ABB RAPID module: hersheyCursiveModule.mod

MODULE hersheyCursiveModule
  ! Character: a
  PROC char_a()
    VAR robtarget pTarget;
    pTarget := refTarget;
    pTarget.trans := [9,17.0,0];
    MoveL pTarget,vSpeed,fine,tTool\WObj:=wWobj;
    Set do_pen;
    pTarget.trans := [8,19.0,0];
    MoveL pTarget,vSpeed,z0,tTool\WObj:=wWobj;
    pTarget.trans := [6,20.0,0];
    MoveL pTarget,vSpeed,z0,tTool\WObj:=wWobj;
    pTarget.trans := [4,20.0,0];
    MoveL pTarget,vSpeed,z0,tTool\WObj:=wWobj;
    pTarget.trans := [2,19.0,0];
    MoveL pTarget,vSpeed,z0,tTool\WObj:=wWobj;
    pTarget.trans := [1,18.0,0];
    MoveL pTarget,vSpeed,z0,tTool\WObj:=wWobj;
    pTarget.trans := [0,16.0,0];
    MoveL pTarget,vSpeed,z0,tTool\WObj:=wWobj;
    pTarget.trans := [0,14.0,0];
    MoveL pTarget,vSpeed,z0,tTool\WObj:=wWobj;
    pTarget.trans := [1,12.0,0];
    MoveL pTarget,vSpeed,z0,tTool\WObj:=wWobj;
    pTarget.trans := [3,11.0,0];
    MoveL pTarget,vSpeed,z0,tTool\WObj:=wWobj;
    pTarget.trans := [5,11.0,0];
    MoveL pTarget,vSpeed,z0,tTool\WObj:=wWobj;
    pTarget.trans := [7,12.0,0];
    MoveL pTarget,vSpeed,z0,tTool\WObj:=wWobj;
    pTarget.trans := [8,14.0,0];
    MoveL pTarget,vSpeed,z0,tTool\WObj:=wWobj;
    pTarget.trans := [10,20.0,0];
    MoveL pTarget,vSpeed,z0,tTool\WObj:=wWobj;
    pTarget.trans := [9,15.0,0];
    MoveL pTarget,vSpeed,z0,tTool\WObj:=wWobj;
    pTarget.trans := [9,12.0,0];
    MoveL pTarget,vSpeed,z0,tTool\WObj:=wWobj;
    pTarget.trans := [10,11.0,0];
    MoveL pTarget,vSpeed,z0,tTool\WObj:=wWobj;
    pTarget.trans := [11,11.0,0];
    MoveL pTarget,vSpeed,z0,tTool\WObj:=wWobj;
    pTarget.trans := [13,12.0,0];
    MoveL pTarget,vSpeed,z0,tTool\WObj:=wWobj;
    pTarget.trans := [14,13.0,0];
    MoveL pTarget,vSpeed,z0,tTool\WObj:=wWobj;
    pTarget.trans := [16,16.0,0];
    MoveL pTarget,vSpeed,fine,tTool\WObj:=wWobj;
    Reset do_pen;
    MoveL RelTool(pTarget,0,0,-2),vSpeed,z0,tTool\WObj:=wWobj;
    wWobj.oframe.trans.x := wWobj.oframe.trans.x + 16;
ENDPROC
  ! Character: b
  PROC char_b()
    VAR robtarget pTarget;
    pTarget := refTarget;
    pTarget.trans := [0,16.0,0];
    MoveL pTarget,vSpeed,fine,tTool\WObj:=wWobj;
    Set do_pen;
    pTarget.trans := [2,19.0,0];
    MoveL pTarget,vSpeed,z0,tTool\WObj:=wWobj;
    pTarget.trans := [5,24.0,0];
    MoveL pTarget,vSpeed,z0,tTool\WObj:=wWobj;
    pTarget.trans := [6,26.0,0];
    MoveL pTarget,vSpeed,z0,tTool\WObj:=wWobj;
    pTarget.trans := [7,29.0,0];
    MoveL pTarget,vSpeed,z0,tTool\WObj:=wWobj;
    pTarget.trans := [7,31.0,0];
    MoveL pTarget,vSpeed,z0,tTool\WObj:=wWobj;
    pTarget.trans := [6,32.0,0];
    MoveL pTarget,vSpeed,z0,tTool\WObj:=wWobj;
    pTarget.trans := [4,31.0,0];
    MoveL pTarget,vSpeed,z0,tTool\WObj:=wWobj;
    pTarget.trans := [3,29.0,0];
    MoveL pTarget,vSpeed,z0,tTool\WObj:=wWobj;
    pTarget.trans := [2,25.0,0];
    MoveL pTarget,vSpeed,z0,tTool\WObj:=wWobj;
    pTarget.trans := [1,18.0,0];
    MoveL pTarget,vSpeed,z0,tTool\WObj:=wWobj;
    pTarget.trans := [1,12.0,0];
    MoveL pTarget,vSpeed,z0,tTool\WObj:=wWobj;
    pTarget.trans := [2,11.0,0];
    MoveL pTarget,vSpeed,z0,tTool\WObj:=wWobj;
    pTarget.trans := [3,11.0,0];
    MoveL pTarget,vSpeed,z0,tTool\WObj:=wWobj;
    pTarget.trans := [5,12.0,0];
    MoveL pTarget,vSpeed,z0,tTool\WObj:=wWobj;
    pTarget.trans := [7,14.0,0];
    MoveL pTarget,vSpeed,z0,tTool\WObj:=wWobj;
    pTarget.trans := [8,17.0,0];
    MoveL pTarget,vSpeed,z0,tTool\WObj:=wWobj;
    pTarget.trans := [8,20.0,0];
    MoveL pTarget,vSpeed,z0,tTool\WObj:=wWobj;
    pTarget.trans := [9,16.0,0];
    MoveL pTarget,vSpeed,z0,tTool\WObj:=wWobj;
    pTarget.trans := [10,15.0,0];
    MoveL pTarget,vSpeed,z0,tTool\WObj:=wWobj;
    pTarget.trans := [12,15.0,0];
    MoveL pTarget,vSpeed,z0,tTool\WObj:=wWobj;
    pTarget.trans := [14,16.0,0];
    MoveL pTarget,vSpeed,fine,tTool\WObj:=wWobj;
    Reset do_pen;
    MoveL RelTool(pTarget,0,0,-2),vSpeed,z0,tTool\WObj:=wWobj;
    wWobj.oframe.trans.x := wWobj.oframe.trans.x + 14;
ENDPROC
  ! Character: c
  PROC char_c()
    VAR robtarget pTarget;
    pTarget := refTarget;
    pTarget.trans := [7,18.0,0];
    MoveL pTarget,vSpeed,fine,tTool\WObj:=wWobj;
    Set do_pen;
    pTarget.trans := [7,19.0,0];
    MoveL pTarget,vSpeed,z0,tTool\WObj:=wWobj;
    pTarget.trans := [6,20.0,0];
    MoveL pTarget,vSpeed,z0,tTool\WObj:=wWobj;
    pTarget.trans := [4,20.0,0];
    MoveL pTarget,vSpeed,z0,tTool\WObj:=wWobj;
    pTarget.trans := [2,19.0,0];
    MoveL pTarget,vSpeed,z0,tTool\WObj:=wWobj;
    pTarget.trans := [1,18.0,0];
    MoveL pTarget,vSpeed,z0,tTool\WObj:=wWobj;
    pTarget.trans := [0,16.0,0];
    MoveL pTarget,vSpeed,z0,tTool\WObj:=wWobj;
    pTarget.trans := [0,14.0,0];
    MoveL pTarget,vSpeed,z0,tTool\WObj:=wWobj;
    pTarget.trans := [1,12.0,0];
    MoveL pTarget,vSpeed,z0,tTool\WObj:=wWobj;
    pTarget.trans := [3,11.0,0];
    MoveL pTarget,vSpeed,z0,tTool\WObj:=wWobj;
    pTarget.trans := [6,11.0,0];
    MoveL pTarget,vSpeed,z0,tTool\WObj:=wWobj;
    pTarget.trans := [9,13.0,0];
    MoveL pTarget,vSpeed,z0,tTool\WObj:=wWobj;
    pTarget.trans := [11,16.0,0];
    MoveL pTarget,vSpeed,fine,tTool\WObj:=wWobj;
    Reset do_pen;
    MoveL RelTool(pTarget,0,0,-2),vSpeed,z0,tTool\WObj:=wWobj;
    wWobj.oframe.trans.x := wWobj.oframe.trans.x + 11;
ENDPROC
  ! Character: d
  PROC char_d()
    VAR robtarget pTarget;
    pTarget := refTarget;
    pTarget.trans := [9,17.0,0];
    MoveL pTarget,vSpeed,fine,tTool\WObj:=wWobj;
    Set do_pen;
    pTarget.trans := [8,19.0,0];
    MoveL pTarget,vSpeed,z0,tTool\WObj:=wWobj;
    pTarget.trans := [6,20.0,0];
    MoveL pTarget,vSpeed,z0,tTool\WObj:=wWobj;
    pTarget.trans := [4,20.0,0];
    MoveL pTarget,vSpeed,z0,tTool\WObj:=wWobj;
    pTarget.trans := [2,19.0,0];
    MoveL pTarget,vSpeed,z0,tTool\WObj:=wWobj;
    pTarget.trans := [1,18.0,0];
    MoveL pTarget,vSpeed,z0,tTool\WObj:=wWobj;
    pTarget.trans := [0,16.0,0];
    MoveL pTarget,vSpeed,z0,tTool\WObj:=wWobj;
    pTarget.trans := [0,14.0,0];
    MoveL pTarget,vSpeed,z0,tTool\WObj:=wWobj;
    pTarget.trans := [1,12.0,0];
    MoveL pTarget,vSpeed,z0,tTool\WObj:=wWobj;
    pTarget.trans := [3,11.0,0];
    MoveL pTarget,vSpeed,z0,tTool\WObj:=wWobj;
    pTarget.trans := [5,11.0,0];
    MoveL pTarget,vSpeed,z0,tTool\WObj:=wWobj;
    pTarget.trans := [7,12.0,0];
    MoveL pTarget,vSpeed,z0,tTool\WObj:=wWobj;
    pTarget.trans := [8,14.0,0];
    MoveL pTarget,vSpeed,z0,tTool\WObj:=wWobj;
    pTarget.trans := [14,32.0,0];
    MoveL pTarget,vSpeed,fine,tTool\WObj:=wWobj;
    Reset do_pen;
    MoveL RelTool(pTarget,0,0,-2),vSpeed,z0,tTool\WObj:=wWobj;
    pTarget.trans := [10,20.0,0];
    MoveL pTarget,vSpeed,fine,tTool\WObj:=wWobj;
    Set do_pen;
    pTarget.trans := [9,15.0,0];
    MoveL pTarget,vSpeed,z0,tTool\WObj:=wWobj;
    pTarget.trans := [9,12.0,0];
    MoveL pTarget,vSpeed,z0,tTool\WObj:=wWobj;
    pTarget.trans := [10,11.0,0];
    MoveL pTarget,vSpeed,z0,tTool\WObj:=wWobj;
    pTarget.trans := [11,11.0,0];
    MoveL pTarget,vSpeed,z0,tTool\WObj:=wWobj;
    pTarget.trans := [13,12.0,0];
    MoveL pTarget,vSpeed,z0,tTool\WObj:=wWobj;
    pTarget.trans := [14,13.0,0];
    MoveL pTarget,vSpeed,z0,tTool\WObj:=wWobj;
    pTarget.trans := [16,16.0,0];
    MoveL pTarget,vSpeed,fine,tTool\WObj:=wWobj;
    Reset do_pen;
    MoveL RelTool(pTarget,0,0,-2),vSpeed,z0,tTool\WObj:=wWobj;
    wWobj.oframe.trans.x := wWobj.oframe.trans.x + 16;
ENDPROC
  ! Character: e
  PROC char_e()
    VAR robtarget pTarget;
    pTarget := refTarget;
    pTarget.trans := [1,13.0,0];
    MoveL pTarget,vSpeed,fine,tTool\WObj:=wWobj;
    Set do_pen;
    pTarget.trans := [3,14.0,0];
    MoveL pTarget,vSpeed,z0,tTool\WObj:=wWobj;
    pTarget.trans := [4,15.0,0];
    MoveL pTarget,vSpeed,z0,tTool\WObj:=wWobj;
    pTarget.trans := [5,17.0,0];
    MoveL pTarget,vSpeed,z0,tTool\WObj:=wWobj;
    pTarget.trans := [5,19.0,0];
    MoveL pTarget,vSpeed,z0,tTool\WObj:=wWobj;
    pTarget.trans := [4,20.0,0];
    MoveL pTarget,vSpeed,z0,tTool\WObj:=wWobj;
    pTarget.trans := [3,20.0,0];
    MoveL pTarget,vSpeed,z0,tTool\WObj:=wWobj;
    pTarget.trans := [1,19.0,0];
    MoveL pTarget,vSpeed,z0,tTool\WObj:=wWobj;
    pTarget.trans := [0,17.0,0];
    MoveL pTarget,vSpeed,z0,tTool\WObj:=wWobj;
    pTarget.trans := [0,14.0,0];
    MoveL pTarget,vSpeed,z0,tTool\WObj:=wWobj;
    pTarget.trans := [1,12.0,0];
    MoveL pTarget,vSpeed,z0,tTool\WObj:=wWobj;
    pTarget.trans := [3,11.0,0];
    MoveL pTarget,vSpeed,z0,tTool\WObj:=wWobj;
    pTarget.trans := [5,11.0,0];
    MoveL pTarget,vSpeed,z0,tTool\WObj:=wWobj;
    pTarget.trans := [7,12.0,0];
    MoveL pTarget,vSpeed,z0,tTool\WObj:=wWobj;
    pTarget.trans := [8,13.0,0];
    MoveL pTarget,vSpeed,z0,tTool\WObj:=wWobj;
    pTarget.trans := [10,16.0,0];
    MoveL pTarget,vSpeed,fine,tTool\WObj:=wWobj;
    Reset do_pen;
    MoveL RelTool(pTarget,0,0,-2),vSpeed,z0,tTool\WObj:=wWobj;
    wWobj.oframe.trans.x := wWobj.oframe.trans.x + 10;
ENDPROC
  ! Character: f
  PROC char_f()
    VAR robtarget pTarget;
    pTarget := refTarget;
    pTarget.trans := [0,16.0,0];
    MoveL pTarget,vSpeed,fine,tTool\WObj:=wWobj;
    Set do_pen;
    pTarget.trans := [4,21.0,0];
    MoveL pTarget,vSpeed,z0,tTool\WObj:=wWobj;
    pTarget.trans := [6,24.0,0];
    MoveL pTarget,vSpeed,z0,tTool\WObj:=wWobj;
    pTarget.trans := [7,26.0,0];
    MoveL pTarget,vSpeed,z0,tTool\WObj:=wWobj;
    pTarget.trans := [8,29.0,0];
    MoveL pTarget,vSpeed,z0,tTool\WObj:=wWobj;
    pTarget.trans := [8,31.0,0];
    MoveL pTarget,vSpeed,z0,tTool\WObj:=wWobj;
    pTarget.trans := [7,32.0,0];
    MoveL pTarget,vSpeed,z0,tTool\WObj:=wWobj;
    pTarget.trans := [5,31.0,0];
    MoveL pTarget,vSpeed,z0,tTool\WObj:=wWobj;
    pTarget.trans := [4,29.0,0];
    MoveL pTarget,vSpeed,z0,tTool\WObj:=wWobj;
    pTarget.trans := [2,21.0,0];
    MoveL pTarget,vSpeed,z0,tTool\WObj:=wWobj;
    pTarget.trans := [-1,12.0,0];
    MoveL pTarget,vSpeed,z0,tTool\WObj:=wWobj;
    pTarget.trans := [-4,5.0,0];
    MoveL pTarget,vSpeed,z0,tTool\WObj:=wWobj;
    pTarget.trans := [-5,2.0,0];
    MoveL pTarget,vSpeed,z0,tTool\WObj:=wWobj;
    pTarget.trans := [-5,0.0,0];
    MoveL pTarget,vSpeed,z0,tTool\WObj:=wWobj;
    pTarget.trans := [-4,-1.0,0];
    MoveL pTarget,vSpeed,z0,tTool\WObj:=wWobj;
    pTarget.trans := [-2,0.0,0];
    MoveL pTarget,vSpeed,z0,tTool\WObj:=wWobj;
    pTarget.trans := [-1,3.0,0];
    MoveL pTarget,vSpeed,z0,tTool\WObj:=wWobj;
    pTarget.trans := [0,12.0,0];
    MoveL pTarget,vSpeed,z0,tTool\WObj:=wWobj;
    pTarget.trans := [1,11.0,0];
    MoveL pTarget,vSpeed,z0,tTool\WObj:=wWobj;
    pTarget.trans := [3,11.0,0];
    MoveL pTarget,vSpeed,z0,tTool\WObj:=wWobj;
    pTarget.trans := [5,12.0,0];
    MoveL pTarget,vSpeed,z0,tTool\WObj:=wWobj;
    pTarget.trans := [6,13.0,0];
    MoveL pTarget,vSpeed,z0,tTool\WObj:=wWobj;
    pTarget.trans := [8,16.0,0];
    MoveL pTarget,vSpeed,fine,tTool\WObj:=wWobj;
    Reset do_pen;
    MoveL RelTool(pTarget,0,0,-2),vSpeed,z0,tTool\WObj:=wWobj;
    wWobj.oframe.trans.x := wWobj.oframe.trans.x + 13;
ENDPROC
  ! Character: g
  PROC char_g()
    VAR robtarget pTarget;
    pTarget := refTarget;
    pTarget.trans := [9,17.0,0];
    MoveL pTarget,vSpeed,fine,tTool\WObj:=wWobj;
    Set do_pen;
    pTarget.trans := [8,19.0,0];
    MoveL pTarget,vSpeed,z0,tTool\WObj:=wWobj;
    pTarget.trans := [6,20.0,0];
    MoveL pTarget,vSpeed,z0,tTool\WObj:=wWobj;
    pTarget.trans := [4,20.0,0];
    MoveL pTarget,vSpeed,z0,tTool\WObj:=wWobj;
    pTarget.trans := [2,19.0,0];
    MoveL pTarget,vSpeed,z0,tTool\WObj:=wWobj;
    pTarget.trans := [1,18.0,0];
    MoveL pTarget,vSpeed,z0,tTool\WObj:=wWobj;
    pTarget.trans := [0,16.0,0];
    MoveL pTarget,vSpeed,z0,tTool\WObj:=wWobj;
    pTarget.trans := [0,14.0,0];
    MoveL pTarget,vSpeed,z0,tTool\WObj:=wWobj;
    pTarget.trans := [1,12.0,0];
    MoveL pTarget,vSpeed,z0,tTool\WObj:=wWobj;
    pTarget.trans := [3,11.0,0];
    MoveL pTarget,vSpeed,z0,tTool\WObj:=wWobj;
    pTarget.trans := [5,11.0,0];
    MoveL pTarget,vSpeed,z0,tTool\WObj:=wWobj;
    pTarget.trans := [7,12.0,0];
    MoveL pTarget,vSpeed,z0,tTool\WObj:=wWobj;
    pTarget.trans := [8,13.0,0];
    MoveL pTarget,vSpeed,fine,tTool\WObj:=wWobj;
    Reset do_pen;
    MoveL RelTool(pTarget,0,0,-2),vSpeed,z0,tTool\WObj:=wWobj;
    pTarget.trans := [10,20.0,0];
    MoveL pTarget,vSpeed,fine,tTool\WObj:=wWobj;
    Set do_pen;
    pTarget.trans := [8,13.0,0];
    MoveL pTarget,vSpeed,z0,tTool\WObj:=wWobj;
    pTarget.trans := [4,2.0,0];
    MoveL pTarget,vSpeed,z0,tTool\WObj:=wWobj;
    pTarget.trans := [3,0.0,0];
    MoveL pTarget,vSpeed,z0,tTool\WObj:=wWobj;
    pTarget.trans := [1,-1.0,0];
    MoveL pTarget,vSpeed,z0,tTool\WObj:=wWobj;
    pTarget.trans := [0,0.0,0];
    MoveL pTarget,vSpeed,z0,tTool\WObj:=wWobj;
    pTarget.trans := [0,2.0,0];
    MoveL pTarget,vSpeed,z0,tTool\WObj:=wWobj;
    pTarget.trans := [1,5.0,0];
    MoveL pTarget,vSpeed,z0,tTool\WObj:=wWobj;
    pTarget.trans := [4,8.0,0];
    MoveL pTarget,vSpeed,z0,tTool\WObj:=wWobj;
    pTarget.trans := [7,10.0,0];
    MoveL pTarget,vSpeed,z0,tTool\WObj:=wWobj;
    pTarget.trans := [9,11.0,0];
    MoveL pTarget,vSpeed,z0,tTool\WObj:=wWobj;
    pTarget.trans := [12,13.0,0];
    MoveL pTarget,vSpeed,z0,tTool\WObj:=wWobj;
    pTarget.trans := [15,16.0,0];
    MoveL pTarget,vSpeed,fine,tTool\WObj:=wWobj;
    Reset do_pen;
    MoveL RelTool(pTarget,0,0,-2),vSpeed,z0,tTool\WObj:=wWobj;
    wWobj.oframe.trans.x := wWobj.oframe.trans.x + 15;
ENDPROC
  ! Character: h
  PROC char_h()
    VAR robtarget pTarget;
    pTarget := refTarget;
    pTarget.trans := [0,16.0,0];
    MoveL pTarget,vSpeed,fine,tTool\WObj:=wWobj;
    Set do_pen;
    pTarget.trans := [2,19.0,0];
    MoveL pTarget,vSpeed,z0,tTool\WObj:=wWobj;
    pTarget.trans := [5,24.0,0];
    MoveL pTarget,vSpeed,z0,tTool\WObj:=wWobj;
    pTarget.trans := [6,26.0,0];
    MoveL pTarget,vSpeed,z0,tTool\WObj:=wWobj;
    pTarget.trans := [7,29.0,0];
    MoveL pTarget,vSpeed,z0,tTool\WObj:=wWobj;
    pTarget.trans := [7,31.0,0];
    MoveL pTarget,vSpeed,z0,tTool\WObj:=wWobj;
    pTarget.trans := [6,32.0,0];
    MoveL pTarget,vSpeed,z0,tTool\WObj:=wWobj;
    pTarget.trans := [4,31.0,0];
    MoveL pTarget,vSpeed,z0,tTool\WObj:=wWobj;
    pTarget.trans := [3,29.0,0];
    MoveL pTarget,vSpeed,z0,tTool\WObj:=wWobj;
    pTarget.trans := [2,25.0,0];
    MoveL pTarget,vSpeed,z0,tTool\WObj:=wWobj;
    pTarget.trans := [1,19.0,0];
    MoveL pTarget,vSpeed,z0,tTool\WObj:=wWobj;
    pTarget.trans := [0,11.0,0];
    MoveL pTarget,vSpeed,fine,tTool\WObj:=wWobj;
    Reset do_pen;
    MoveL RelTool(pTarget,0,0,-2),vSpeed,z0,tTool\WObj:=wWobj;
    pTarget.trans := [0,11.0,0];
    MoveL pTarget,vSpeed,fine,tTool\WObj:=wWobj;
    Set do_pen;
    pTarget.trans := [1,14.0,0];
    MoveL pTarget,vSpeed,z0,tTool\WObj:=wWobj;
    pTarget.trans := [2,16.0,0];
    MoveL pTarget,vSpeed,z0,tTool\WObj:=wWobj;
    pTarget.trans := [4,19.0,0];
    MoveL pTarget,vSpeed,z0,tTool\WObj:=wWobj;
    pTarget.trans := [6,20.0,0];
    MoveL pTarget,vSpeed,z0,tTool\WObj:=wWobj;
    pTarget.trans := [8,20.0,0];
    MoveL pTarget,vSpeed,z0,tTool\WObj:=wWobj;
    pTarget.trans := [9,19.0,0];
    MoveL pTarget,vSpeed,z0,tTool\WObj:=wWobj;
    pTarget.trans := [9,17.0,0];
    MoveL pTarget,vSpeed,z0,tTool\WObj:=wWobj;
    pTarget.trans := [8,14.0,0];
    MoveL pTarget,vSpeed,z0,tTool\WObj:=wWobj;
    pTarget.trans := [8,12.0,0];
    MoveL pTarget,vSpeed,z0,tTool\WObj:=wWobj;
    pTarget.trans := [9,11.0,0];
    MoveL pTarget,vSpeed,z0,tTool\WObj:=wWobj;
    pTarget.trans := [10,11.0,0];
    MoveL pTarget,vSpeed,z0,tTool\WObj:=wWobj;
    pTarget.trans := [12,12.0,0];
    MoveL pTarget,vSpeed,z0,tTool\WObj:=wWobj;
    pTarget.trans := [13,13.0,0];
    MoveL pTarget,vSpeed,z0,tTool\WObj:=wWobj;
    pTarget.trans := [15,16.0,0];
    MoveL pTarget,vSpeed,fine,tTool\WObj:=wWobj;
    Reset do_pen;
    MoveL RelTool(pTarget,0,0,-2),vSpeed,z0,tTool\WObj:=wWobj;
    wWobj.oframe.trans.x := wWobj.oframe.trans.x + 15;
ENDPROC
  ! Character: i
  PROC char_i()
    VAR robtarget pTarget;
    pTarget := refTarget;
    pTarget.trans := [3,25.0,0];
    MoveL pTarget,vSpeed,fine,tTool\WObj:=wWobj;
    Set do_pen;
    pTarget.trans := [3,24.0,0];
    MoveL pTarget,vSpeed,z0,tTool\WObj:=wWobj;
    pTarget.trans := [4,24.0,0];
    MoveL pTarget,vSpeed,z0,tTool\WObj:=wWobj;
    pTarget.trans := [4,25.0,0];
    MoveL pTarget,vSpeed,z0,tTool\WObj:=wWobj;
    pTarget.trans := [3,25.0,0];
    MoveL pTarget,vSpeed,fine,tTool\WObj:=wWobj;
    Reset do_pen;
    MoveL RelTool(pTarget,0,0,-2),vSpeed,z0,tTool\WObj:=wWobj;
    pTarget.trans := [0,16.0,0];
    MoveL pTarget,vSpeed,fine,tTool\WObj:=wWobj;
    Set do_pen;
    pTarget.trans := [2,20.0,0];
    MoveL pTarget,vSpeed,z0,tTool\WObj:=wWobj;
    pTarget.trans := [0,14.0,0];
    MoveL pTarget,vSpeed,z0,tTool\WObj:=wWobj;
    pTarget.trans := [0,12.0,0];
    MoveL pTarget,vSpeed,z0,tTool\WObj:=wWobj;
    pTarget.trans := [1,11.0,0];
    MoveL pTarget,vSpeed,z0,tTool\WObj:=wWobj;
    pTarget.trans := [2,11.0,0];
    MoveL pTarget,vSpeed,z0,tTool\WObj:=wWobj;
    pTarget.trans := [4,12.0,0];
    MoveL pTarget,vSpeed,z0,tTool\WObj:=wWobj;
    pTarget.trans := [5,13.0,0];
    MoveL pTarget,vSpeed,z0,tTool\WObj:=wWobj;
    pTarget.trans := [7,16.0,0];
    MoveL pTarget,vSpeed,fine,tTool\WObj:=wWobj;
    Reset do_pen;
    MoveL RelTool(pTarget,0,0,-2),vSpeed,z0,tTool\WObj:=wWobj;
    wWobj.oframe.trans.x := wWobj.oframe.trans.x + 7;
ENDPROC
  ! Character: j
  PROC char_j()
    VAR robtarget pTarget;
    pTarget := refTarget;
    pTarget.trans := [3,25.0,0];
    MoveL pTarget,vSpeed,fine,tTool\WObj:=wWobj;
    Set do_pen;
    pTarget.trans := [3,24.0,0];
    MoveL pTarget,vSpeed,z0,tTool\WObj:=wWobj;
    pTarget.trans := [4,24.0,0];
    MoveL pTarget,vSpeed,z0,tTool\WObj:=wWobj;
    pTarget.trans := [4,25.0,0];
    MoveL pTarget,vSpeed,z0,tTool\WObj:=wWobj;
    pTarget.trans := [3,25.0,0];
    MoveL pTarget,vSpeed,fine,tTool\WObj:=wWobj;
    Reset do_pen;
    MoveL RelTool(pTarget,0,0,-2),vSpeed,z0,tTool\WObj:=wWobj;
    pTarget.trans := [0,16.0,0];
    MoveL pTarget,vSpeed,fine,tTool\WObj:=wWobj;
    Set do_pen;
    pTarget.trans := [2,20.0,0];
    MoveL pTarget,vSpeed,z0,tTool\WObj:=wWobj;
    pTarget.trans := [-4,2.0,0];
    MoveL pTarget,vSpeed,z0,tTool\WObj:=wWobj;
    pTarget.trans := [-5,0.0,0];
    MoveL pTarget,vSpeed,z0,tTool\WObj:=wWobj;
    pTarget.trans := [-7,-1.0,0];
    MoveL pTarget,vSpeed,z0,tTool\WObj:=wWobj;
    pTarget.trans := [-8,0.0,0];
    MoveL pTarget,vSpeed,z0,tTool\WObj:=wWobj;
    pTarget.trans := [-8,2.0,0];
    MoveL pTarget,vSpeed,z0,tTool\WObj:=wWobj;
    pTarget.trans := [-7,5.0,0];
    MoveL pTarget,vSpeed,z0,tTool\WObj:=wWobj;
    pTarget.trans := [-4,8.0,0];
    MoveL pTarget,vSpeed,z0,tTool\WObj:=wWobj;
    pTarget.trans := [-1,10.0,0];
    MoveL pTarget,vSpeed,z0,tTool\WObj:=wWobj;
    pTarget.trans := [1,11.0,0];
    MoveL pTarget,vSpeed,z0,tTool\WObj:=wWobj;
    pTarget.trans := [4,13.0,0];
    MoveL pTarget,vSpeed,z0,tTool\WObj:=wWobj;
    pTarget.trans := [7,16.0,0];
    MoveL pTarget,vSpeed,fine,tTool\WObj:=wWobj;
    Reset do_pen;
    MoveL RelTool(pTarget,0,0,-2),vSpeed,z0,tTool\WObj:=wWobj;
    wWobj.oframe.trans.x := wWobj.oframe.trans.x + 15;
ENDPROC
  ! Character: k
  PROC char_k()
    VAR robtarget pTarget;
    pTarget := refTarget;
    pTarget.trans := [0,16.0,0];
    MoveL pTarget,vSpeed,fine,tTool\WObj:=wWobj;
    Set do_pen;
    pTarget.trans := [2,19.0,0];
    MoveL pTarget,vSpeed,z0,tTool\WObj:=wWobj;
    pTarget.trans := [5,24.0,0];
    MoveL pTarget,vSpeed,z0,tTool\WObj:=wWobj;
    pTarget.trans := [6,26.0,0];
    MoveL pTarget,vSpeed,z0,tTool\WObj:=wWobj;
    pTarget.trans := [7,29.0,0];
    MoveL pTarget,vSpeed,z0,tTool\WObj:=wWobj;
    pTarget.trans := [7,31.0,0];
    MoveL pTarget,vSpeed,z0,tTool\WObj:=wWobj;
    pTarget.trans := [6,32.0,0];
    MoveL pTarget,vSpeed,z0,tTool\WObj:=wWobj;
    pTarget.trans := [4,31.0,0];
    MoveL pTarget,vSpeed,z0,tTool\WObj:=wWobj;
    pTarget.trans := [3,29.0,0];
    MoveL pTarget,vSpeed,z0,tTool\WObj:=wWobj;
    pTarget.trans := [2,25.0,0];
    MoveL pTarget,vSpeed,z0,tTool\WObj:=wWobj;
    pTarget.trans := [1,19.0,0];
    MoveL pTarget,vSpeed,z0,tTool\WObj:=wWobj;
    pTarget.trans := [0,11.0,0];
    MoveL pTarget,vSpeed,fine,tTool\WObj:=wWobj;
    Reset do_pen;
    MoveL RelTool(pTarget,0,0,-2),vSpeed,z0,tTool\WObj:=wWobj;
    pTarget.trans := [0,11.0,0];
    MoveL pTarget,vSpeed,fine,tTool\WObj:=wWobj;
    Set do_pen;
    pTarget.trans := [1,14.0,0];
    MoveL pTarget,vSpeed,z0,tTool\WObj:=wWobj;
    pTarget.trans := [2,16.0,0];
    MoveL pTarget,vSpeed,z0,tTool\WObj:=wWobj;
    pTarget.trans := [4,19.0,0];
    MoveL pTarget,vSpeed,z0,tTool\WObj:=wWobj;
    pTarget.trans := [6,20.0,0];
    MoveL pTarget,vSpeed,z0,tTool\WObj:=wWobj;
    pTarget.trans := [8,20.0,0];
    MoveL pTarget,vSpeed,z0,tTool\WObj:=wWobj;
    pTarget.trans := [9,19.0,0];
    MoveL pTarget,vSpeed,z0,tTool\WObj:=wWobj;
    pTarget.trans := [9,17.0,0];
    MoveL pTarget,vSpeed,z0,tTool\WObj:=wWobj;
    pTarget.trans := [7,16.0,0];
    MoveL pTarget,vSpeed,z0,tTool\WObj:=wWobj;
    pTarget.trans := [4,16.0,0];
    MoveL pTarget,vSpeed,fine,tTool\WObj:=wWobj;
    Reset do_pen;
    MoveL RelTool(pTarget,0,0,-2),vSpeed,z0,tTool\WObj:=wWobj;
    pTarget.trans := [4,16.0,0];
    MoveL pTarget,vSpeed,fine,tTool\WObj:=wWobj;
    Set do_pen;
    pTarget.trans := [6,15.0,0];
    MoveL pTarget,vSpeed,z0,tTool\WObj:=wWobj;
    pTarget.trans := [7,12.0,0];
    MoveL pTarget,vSpeed,z0,tTool\WObj:=wWobj;
    pTarget.trans := [8,11.0,0];
    MoveL pTarget,vSpeed,z0,tTool\WObj:=wWobj;
    pTarget.trans := [9,11.0,0];
    MoveL pTarget,vSpeed,z0,tTool\WObj:=wWobj;
    pTarget.trans := [11,12.0,0];
    MoveL pTarget,vSpeed,z0,tTool\WObj:=wWobj;
    pTarget.trans := [12,13.0,0];
    MoveL pTarget,vSpeed,z0,tTool\WObj:=wWobj;
    pTarget.trans := [14,16.0,0];
    MoveL pTarget,vSpeed,fine,tTool\WObj:=wWobj;
    Reset do_pen;
    MoveL RelTool(pTarget,0,0,-2),vSpeed,z0,tTool\WObj:=wWobj;
    wWobj.oframe.trans.x := wWobj.oframe.trans.x + 14;
ENDPROC
  ! Character: l
  PROC char_l()
    VAR robtarget pTarget;
    pTarget := refTarget;
    pTarget.trans := [0,16.0,0];
    MoveL pTarget,vSpeed,fine,tTool\WObj:=wWobj;
    Set do_pen;
    pTarget.trans := [2,19.0,0];
    MoveL pTarget,vSpeed,z0,tTool\WObj:=wWobj;
    pTarget.trans := [5,24.0,0];
    MoveL pTarget,vSpeed,z0,tTool\WObj:=wWobj;
    pTarget.trans := [6,26.0,0];
    MoveL pTarget,vSpeed,z0,tTool\WObj:=wWobj;
    pTarget.trans := [7,29.0,0];
    MoveL pTarget,vSpeed,z0,tTool\WObj:=wWobj;
    pTarget.trans := [7,31.0,0];
    MoveL pTarget,vSpeed,z0,tTool\WObj:=wWobj;
    pTarget.trans := [6,32.0,0];
    MoveL pTarget,vSpeed,z0,tTool\WObj:=wWobj;
    pTarget.trans := [4,31.0,0];
    MoveL pTarget,vSpeed,z0,tTool\WObj:=wWobj;
    pTarget.trans := [3,29.0,0];
    MoveL pTarget,vSpeed,z0,tTool\WObj:=wWobj;
    pTarget.trans := [2,25.0,0];
    MoveL pTarget,vSpeed,z0,tTool\WObj:=wWobj;
    pTarget.trans := [1,18.0,0];
    MoveL pTarget,vSpeed,z0,tTool\WObj:=wWobj;
    pTarget.trans := [1,12.0,0];
    MoveL pTarget,vSpeed,z0,tTool\WObj:=wWobj;
    pTarget.trans := [2,11.0,0];
    MoveL pTarget,vSpeed,z0,tTool\WObj:=wWobj;
    pTarget.trans := [3,11.0,0];
    MoveL pTarget,vSpeed,z0,tTool\WObj:=wWobj;
    pTarget.trans := [5,12.0,0];
    MoveL pTarget,vSpeed,z0,tTool\WObj:=wWobj;
    pTarget.trans := [6,13.0,0];
    MoveL pTarget,vSpeed,z0,tTool\WObj:=wWobj;
    pTarget.trans := [8,16.0,0];
    MoveL pTarget,vSpeed,fine,tTool\WObj:=wWobj;
    Reset do_pen;
    MoveL RelTool(pTarget,0,0,-2),vSpeed,z0,tTool\WObj:=wWobj;
    wWobj.oframe.trans.x := wWobj.oframe.trans.x + 8;
ENDPROC
  ! Character: m
  PROC char_m()
    VAR robtarget pTarget;
    pTarget := refTarget;
    pTarget.trans := [0,16.0,0];
    MoveL pTarget,vSpeed,fine,tTool\WObj:=wWobj;
    Set do_pen;
    pTarget.trans := [2,19.0,0];
    MoveL pTarget,vSpeed,z0,tTool\WObj:=wWobj;
    pTarget.trans := [4,20.0,0];
    MoveL pTarget,vSpeed,z0,tTool\WObj:=wWobj;
    pTarget.trans := [5,19.0,0];
    MoveL pTarget,vSpeed,z0,tTool\WObj:=wWobj;
    pTarget.trans := [5,18.0,0];
    MoveL pTarget,vSpeed,z0,tTool\WObj:=wWobj;
    pTarget.trans := [4,14.0,0];
    MoveL pTarget,vSpeed,z0,tTool\WObj:=wWobj;
    pTarget.trans := [3,11.0,0];
    MoveL pTarget,vSpeed,fine,tTool\WObj:=wWobj;
    Reset do_pen;
    MoveL RelTool(pTarget,0,0,-2),vSpeed,z0,tTool\WObj:=wWobj;
    pTarget.trans := [4,14.0,0];
    MoveL pTarget,vSpeed,fine,tTool\WObj:=wWobj;
    Set do_pen;
    pTarget.trans := [5,16.0,0];
    MoveL pTarget,vSpeed,z0,tTool\WObj:=wWobj;
    pTarget.trans := [7,19.0,0];
    MoveL pTarget,vSpeed,z0,tTool\WObj:=wWobj;
    pTarget.trans := [9,20.0,0];
    MoveL pTarget,vSpeed,z0,tTool\WObj:=wWobj;
    pTarget.trans := [11,20.0,0];
    MoveL pTarget,vSpeed,z0,tTool\WObj:=wWobj;
    pTarget.trans := [12,19.0,0];
    MoveL pTarget,vSpeed,z0,tTool\WObj:=wWobj;
    pTarget.trans := [12,18.0,0];
    MoveL pTarget,vSpeed,z0,tTool\WObj:=wWobj;
    pTarget.trans := [11,14.0,0];
    MoveL pTarget,vSpeed,z0,tTool\WObj:=wWobj;
    pTarget.trans := [10,11.0,0];
    MoveL pTarget,vSpeed,fine,tTool\WObj:=wWobj;
    Reset do_pen;
    MoveL RelTool(pTarget,0,0,-2),vSpeed,z0,tTool\WObj:=wWobj;
    pTarget.trans := [11,14.0,0];
    MoveL pTarget,vSpeed,fine,tTool\WObj:=wWobj;
    Set do_pen;
    pTarget.trans := [12,16.0,0];
    MoveL pTarget,vSpeed,z0,tTool\WObj:=wWobj;
    pTarget.trans := [14,19.0,0];
    MoveL pTarget,vSpeed,z0,tTool\WObj:=wWobj;
    pTarget.trans := [16,20.0,0];
    MoveL pTarget,vSpeed,z0,tTool\WObj:=wWobj;
    pTarget.trans := [18,20.0,0];
    MoveL pTarget,vSpeed,z0,tTool\WObj:=wWobj;
    pTarget.trans := [19,19.0,0];
    MoveL pTarget,vSpeed,z0,tTool\WObj:=wWobj;
    pTarget.trans := [19,17.0,0];
    MoveL pTarget,vSpeed,z0,tTool\WObj:=wWobj;
    pTarget.trans := [18,14.0,0];
    MoveL pTarget,vSpeed,z0,tTool\WObj:=wWobj;
    pTarget.trans := [18,12.0,0];
    MoveL pTarget,vSpeed,z0,tTool\WObj:=wWobj;
    pTarget.trans := [19,11.0,0];
    MoveL pTarget,vSpeed,z0,tTool\WObj:=wWobj;
    pTarget.trans := [20,11.0,0];
    MoveL pTarget,vSpeed,z0,tTool\WObj:=wWobj;
    pTarget.trans := [22,12.0,0];
    MoveL pTarget,vSpeed,z0,tTool\WObj:=wWobj;
    pTarget.trans := [23,13.0,0];
    MoveL pTarget,vSpeed,z0,tTool\WObj:=wWobj;
    pTarget.trans := [25,16.0,0];
    MoveL pTarget,vSpeed,fine,tTool\WObj:=wWobj;
    Reset do_pen;
    MoveL RelTool(pTarget,0,0,-2),vSpeed,z0,tTool\WObj:=wWobj;
    wWobj.oframe.trans.x := wWobj.oframe.trans.x + 25;
ENDPROC
  ! Character: n
  PROC char_n()
    VAR robtarget pTarget;
    pTarget := refTarget;
    pTarget.trans := [0,16.0,0];
    MoveL pTarget,vSpeed,fine,tTool\WObj:=wWobj;
    Set do_pen;
    pTarget.trans := [2,19.0,0];
    MoveL pTarget,vSpeed,z0,tTool\WObj:=wWobj;
    pTarget.trans := [4,20.0,0];
    MoveL pTarget,vSpeed,z0,tTool\WObj:=wWobj;
    pTarget.trans := [5,19.0,0];
    MoveL pTarget,vSpeed,z0,tTool\WObj:=wWobj;
    pTarget.trans := [5,18.0,0];
    MoveL pTarget,vSpeed,z0,tTool\WObj:=wWobj;
    pTarget.trans := [4,14.0,0];
    MoveL pTarget,vSpeed,z0,tTool\WObj:=wWobj;
    pTarget.trans := [3,11.0,0];
    MoveL pTarget,vSpeed,fine,tTool\WObj:=wWobj;
    Reset do_pen;
    MoveL RelTool(pTarget,0,0,-2),vSpeed,z0,tTool\WObj:=wWobj;
    pTarget.trans := [4,14.0,0];
    MoveL pTarget,vSpeed,fine,tTool\WObj:=wWobj;
    Set do_pen;
    pTarget.trans := [5,16.0,0];
    MoveL pTarget,vSpeed,z0,tTool\WObj:=wWobj;
    pTarget.trans := [7,19.0,0];
    MoveL pTarget,vSpeed,z0,tTool\WObj:=wWobj;
    pTarget.trans := [9,20.0,0];
    MoveL pTarget,vSpeed,z0,tTool\WObj:=wWobj;
    pTarget.trans := [11,20.0,0];
    MoveL pTarget,vSpeed,z0,tTool\WObj:=wWobj;
    pTarget.trans := [12,19.0,0];
    MoveL pTarget,vSpeed,z0,tTool\WObj:=wWobj;
    pTarget.trans := [12,17.0,0];
    MoveL pTarget,vSpeed,z0,tTool\WObj:=wWobj;
    pTarget.trans := [11,14.0,0];
    MoveL pTarget,vSpeed,z0,tTool\WObj:=wWobj;
    pTarget.trans := [11,12.0,0];
    MoveL pTarget,vSpeed,z0,tTool\WObj:=wWobj;
    pTarget.trans := [12,11.0,0];
    MoveL pTarget,vSpeed,z0,tTool\WObj:=wWobj;
    pTarget.trans := [13,11.0,0];
    MoveL pTarget,vSpeed,z0,tTool\WObj:=wWobj;
    pTarget.trans := [15,12.0,0];
    MoveL pTarget,vSpeed,z0,tTool\WObj:=wWobj;
    pTarget.trans := [16,13.0,0];
    MoveL pTarget,vSpeed,z0,tTool\WObj:=wWobj;
    pTarget.trans := [18,16.0,0];
    MoveL pTarget,vSpeed,fine,tTool\WObj:=wWobj;
    Reset do_pen;
    MoveL RelTool(pTarget,0,0,-2),vSpeed,z0,tTool\WObj:=wWobj;
    wWobj.oframe.trans.x := wWobj.oframe.trans.x + 18;
ENDPROC
  ! Character: o
  PROC char_o()
    VAR robtarget pTarget;
    pTarget := refTarget;
    pTarget.trans := [6,20.0,0];
    MoveL pTarget,vSpeed,fine,tTool\WObj:=wWobj;
    Set do_pen;
    pTarget.trans := [4,20.0,0];
    MoveL pTarget,vSpeed,z0,tTool\WObj:=wWobj;
    pTarget.trans := [2,19.0,0];
    MoveL pTarget,vSpeed,z0,tTool\WObj:=wWobj;
    pTarget.trans := [1,18.0,0];
    MoveL pTarget,vSpeed,z0,tTool\WObj:=wWobj;
    pTarget.trans := [0,16.0,0];
    MoveL pTarget,vSpeed,z0,tTool\WObj:=wWobj;
    pTarget.trans := [0,14.0,0];
    MoveL pTarget,vSpeed,z0,tTool\WObj:=wWobj;
    pTarget.trans := [1,12.0,0];
    MoveL pTarget,vSpeed,z0,tTool\WObj:=wWobj;
    pTarget.trans := [3,11.0,0];
    MoveL pTarget,vSpeed,z0,tTool\WObj:=wWobj;
    pTarget.trans := [5,11.0,0];
    MoveL pTarget,vSpeed,z0,tTool\WObj:=wWobj;
    pTarget.trans := [7,12.0,0];
    MoveL pTarget,vSpeed,z0,tTool\WObj:=wWobj;
    pTarget.trans := [8,13.0,0];
    MoveL pTarget,vSpeed,z0,tTool\WObj:=wWobj;
    pTarget.trans := [9,15.0,0];
    MoveL pTarget,vSpeed,z0,tTool\WObj:=wWobj;
    pTarget.trans := [9,17.0,0];
    MoveL pTarget,vSpeed,z0,tTool\WObj:=wWobj;
    pTarget.trans := [8,19.0,0];
    MoveL pTarget,vSpeed,z0,tTool\WObj:=wWobj;
    pTarget.trans := [6,20.0,0];
    MoveL pTarget,vSpeed,z0,tTool\WObj:=wWobj;
    pTarget.trans := [5,19.0,0];
    MoveL pTarget,vSpeed,z0,tTool\WObj:=wWobj;
    pTarget.trans := [5,17.0,0];
    MoveL pTarget,vSpeed,z0,tTool\WObj:=wWobj;
    pTarget.trans := [6,15.0,0];
    MoveL pTarget,vSpeed,z0,tTool\WObj:=wWobj;
    pTarget.trans := [8,14.0,0];
    MoveL pTarget,vSpeed,z0,tTool\WObj:=wWobj;
    pTarget.trans := [11,14.0,0];
    MoveL pTarget,vSpeed,z0,tTool\WObj:=wWobj;
    pTarget.trans := [13,15.0,0];
    MoveL pTarget,vSpeed,z0,tTool\WObj:=wWobj;
    pTarget.trans := [14,16.0,0];
    MoveL pTarget,vSpeed,fine,tTool\WObj:=wWobj;
    Reset do_pen;
    MoveL RelTool(pTarget,0,0,-2),vSpeed,z0,tTool\WObj:=wWobj;
    wWobj.oframe.trans.x := wWobj.oframe.trans.x + 14;
ENDPROC
  ! Character: p
  PROC char_p()
    VAR robtarget pTarget;
    pTarget := refTarget;
    pTarget.trans := [0,16.0,0];
    MoveL pTarget,vSpeed,fine,tTool\WObj:=wWobj;
    Set do_pen;
    pTarget.trans := [2,19.0,0];
    MoveL pTarget,vSpeed,z0,tTool\WObj:=wWobj;
    pTarget.trans := [3,21.0,0];
    MoveL pTarget,vSpeed,z0,tTool\WObj:=wWobj;
    pTarget.trans := [2,17.0,0];
    MoveL pTarget,vSpeed,z0,tTool\WObj:=wWobj;
    pTarget.trans := [-4,-1.0,0];
    MoveL pTarget,vSpeed,fine,tTool\WObj:=wWobj;
    Reset do_pen;
    MoveL RelTool(pTarget,0,0,-2),vSpeed,z0,tTool\WObj:=wWobj;
    pTarget.trans := [2,17.0,0];
    MoveL pTarget,vSpeed,fine,tTool\WObj:=wWobj;
    Set do_pen;
    pTarget.trans := [3,19.0,0];
    MoveL pTarget,vSpeed,z0,tTool\WObj:=wWobj;
    pTarget.trans := [5,20.0,0];
    MoveL pTarget,vSpeed,z0,tTool\WObj:=wWobj;
    pTarget.trans := [7,20.0,0];
    MoveL pTarget,vSpeed,z0,tTool\WObj:=wWobj;
    pTarget.trans := [9,19.0,0];
    MoveL pTarget,vSpeed,z0,tTool\WObj:=wWobj;
    pTarget.trans := [10,17.0,0];
    MoveL pTarget,vSpeed,z0,tTool\WObj:=wWobj;
    pTarget.trans := [10,15.0,0];
    MoveL pTarget,vSpeed,z0,tTool\WObj:=wWobj;
    pTarget.trans := [9,13.0,0];
    MoveL pTarget,vSpeed,z0,tTool\WObj:=wWobj;
    pTarget.trans := [8,12.0,0];
    MoveL pTarget,vSpeed,z0,tTool\WObj:=wWobj;
    pTarget.trans := [6,11.0,0];
    MoveL pTarget,vSpeed,fine,tTool\WObj:=wWobj;
    Reset do_pen;
    MoveL RelTool(pTarget,0,0,-2),vSpeed,z0,tTool\WObj:=wWobj;
    pTarget.trans := [2,12.0,0];
    MoveL pTarget,vSpeed,fine,tTool\WObj:=wWobj;
    Set do_pen;
    pTarget.trans := [4,11.0,0];
    MoveL pTarget,vSpeed,z0,tTool\WObj:=wWobj;
    pTarget.trans := [7,11.0,0];
    MoveL pTarget,vSpeed,z0,tTool\WObj:=wWobj;
    pTarget.trans := [10,12.0,0];
    MoveL pTarget,vSpeed,z0,tTool\WObj:=wWobj;
    pTarget.trans := [12,13.0,0];
    MoveL pTarget,vSpeed,z0,tTool\WObj:=wWobj;
    pTarget.trans := [15,16.0,0];
    MoveL pTarget,vSpeed,fine,tTool\WObj:=wWobj;
    Reset do_pen;
    MoveL RelTool(pTarget,0,0,-2),vSpeed,z0,tTool\WObj:=wWobj;
    wWobj.oframe.trans.x := wWobj.oframe.trans.x + 19;
ENDPROC
  ! Character: q
  PROC char_q()
    VAR robtarget pTarget;
    pTarget := refTarget;
    pTarget.trans := [9,17.0,0];
    MoveL pTarget,vSpeed,fine,tTool\WObj:=wWobj;
    Set do_pen;
    pTarget.trans := [8,19.0,0];
    MoveL pTarget,vSpeed,z0,tTool\WObj:=wWobj;
    pTarget.trans := [6,20.0,0];
    MoveL pTarget,vSpeed,z0,tTool\WObj:=wWobj;
    pTarget.trans := [4,20.0,0];
    MoveL pTarget,vSpeed,z0,tTool\WObj:=wWobj;
    pTarget.trans := [2,19.0,0];
    MoveL pTarget,vSpeed,z0,tTool\WObj:=wWobj;
    pTarget.trans := [1,18.0,0];
    MoveL pTarget,vSpeed,z0,tTool\WObj:=wWobj;
    pTarget.trans := [0,16.0,0];
    MoveL pTarget,vSpeed,z0,tTool\WObj:=wWobj;
    pTarget.trans := [0,14.0,0];
    MoveL pTarget,vSpeed,z0,tTool\WObj:=wWobj;
    pTarget.trans := [1,12.0,0];
    MoveL pTarget,vSpeed,z0,tTool\WObj:=wWobj;
    pTarget.trans := [3,11.0,0];
    MoveL pTarget,vSpeed,z0,tTool\WObj:=wWobj;
    pTarget.trans := [5,11.0,0];
    MoveL pTarget,vSpeed,z0,tTool\WObj:=wWobj;
    pTarget.trans := [7,12.0,0];
    MoveL pTarget,vSpeed,fine,tTool\WObj:=wWobj;
    Reset do_pen;
    MoveL RelTool(pTarget,0,0,-2),vSpeed,z0,tTool\WObj:=wWobj;
    pTarget.trans := [10,20.0,0];
    MoveL pTarget,vSpeed,fine,tTool\WObj:=wWobj;
    Set do_pen;
    pTarget.trans := [9,17.0,0];
    MoveL pTarget,vSpeed,z0,tTool\WObj:=wWobj;
    pTarget.trans := [7,12.0,0];
    MoveL pTarget,vSpeed,z0,tTool\WObj:=wWobj;
    pTarget.trans := [4,5.0,0];
    MoveL pTarget,vSpeed,z0,tTool\WObj:=wWobj;
    pTarget.trans := [3,2.0,0];
    MoveL pTarget,vSpeed,z0,tTool\WObj:=wWobj;
    pTarget.trans := [3,0.0,0];
    MoveL pTarget,vSpeed,z0,tTool\WObj:=wWobj;
    pTarget.trans := [4,-1.0,0];
    MoveL pTarget,vSpeed,z0,tTool\WObj:=wWobj;
    pTarget.trans := [6,0.0,0];
    MoveL pTarget,vSpeed,z0,tTool\WObj:=wWobj;
    pTarget.trans := [7,3.0,0];
    MoveL pTarget,vSpeed,z0,tTool\WObj:=wWobj;
    pTarget.trans := [7,10.0,0];
    MoveL pTarget,vSpeed,z0,tTool\WObj:=wWobj;
    pTarget.trans := [9,11.0,0];
    MoveL pTarget,vSpeed,z0,tTool\WObj:=wWobj;
    pTarget.trans := [12,13.0,0];
    MoveL pTarget,vSpeed,z0,tTool\WObj:=wWobj;
    pTarget.trans := [15,16.0,0];
    MoveL pTarget,vSpeed,fine,tTool\WObj:=wWobj;
    Reset do_pen;
    MoveL RelTool(pTarget,0,0,-2),vSpeed,z0,tTool\WObj:=wWobj;
    wWobj.oframe.trans.x := wWobj.oframe.trans.x + 15;
ENDPROC
  ! Character: r
  PROC char_r()
    VAR robtarget pTarget;
    pTarget := refTarget;
    pTarget.trans := [0,16.0,0];
    MoveL pTarget,vSpeed,fine,tTool\WObj:=wWobj;
    Set do_pen;
    pTarget.trans := [2,19.0,0];
    MoveL pTarget,vSpeed,z0,tTool\WObj:=wWobj;
    pTarget.trans := [3,21.0,0];
    MoveL pTarget,vSpeed,z0,tTool\WObj:=wWobj;
    pTarget.trans := [3,19.0,0];
    MoveL pTarget,vSpeed,z0,tTool\WObj:=wWobj;
    pTarget.trans := [6,19.0,0];
    MoveL pTarget,vSpeed,z0,tTool\WObj:=wWobj;
    pTarget.trans := [7,18.0,0];
    MoveL pTarget,vSpeed,z0,tTool\WObj:=wWobj;
    pTarget.trans := [7,16.0,0];
    MoveL pTarget,vSpeed,z0,tTool\WObj:=wWobj;
    pTarget.trans := [6,13.0,0];
    MoveL pTarget,vSpeed,z0,tTool\WObj:=wWobj;
    pTarget.trans := [6,12.0,0];
    MoveL pTarget,vSpeed,z0,tTool\WObj:=wWobj;
    pTarget.trans := [7,11.0,0];
    MoveL pTarget,vSpeed,z0,tTool\WObj:=wWobj;
    pTarget.trans := [8,11.0,0];
    MoveL pTarget,vSpeed,z0,tTool\WObj:=wWobj;
    pTarget.trans := [10,12.0,0];
    MoveL pTarget,vSpeed,z0,tTool\WObj:=wWobj;
    pTarget.trans := [11,13.0,0];
    MoveL pTarget,vSpeed,z0,tTool\WObj:=wWobj;
    pTarget.trans := [13,16.0,0];
    MoveL pTarget,vSpeed,fine,tTool\WObj:=wWobj;
    Reset do_pen;
    MoveL RelTool(pTarget,0,0,-2),vSpeed,z0,tTool\WObj:=wWobj;
    wWobj.oframe.trans.x := wWobj.oframe.trans.x + 13;
ENDPROC
  ! Character: s
  PROC char_s()
    VAR robtarget pTarget;
    pTarget := refTarget;
    pTarget.trans := [0,16.0,0];
    MoveL pTarget,vSpeed,fine,tTool\WObj:=wWobj;
    Set do_pen;
    pTarget.trans := [2,19.0,0];
    MoveL pTarget,vSpeed,z0,tTool\WObj:=wWobj;
    pTarget.trans := [3,21.0,0];
    MoveL pTarget,vSpeed,z0,tTool\WObj:=wWobj;
    pTarget.trans := [3,19.0,0];
    MoveL pTarget,vSpeed,z0,tTool\WObj:=wWobj;
    pTarget.trans := [5,16.0,0];
    MoveL pTarget,vSpeed,z0,tTool\WObj:=wWobj;
    pTarget.trans := [6,14.0,0];
    MoveL pTarget,vSpeed,z0,tTool\WObj:=wWobj;
    pTarget.trans := [6,12.0,0];
    MoveL pTarget,vSpeed,z0,tTool\WObj:=wWobj;
    pTarget.trans := [4,11.0,0];
    MoveL pTarget,vSpeed,fine,tTool\WObj:=wWobj;
    Reset do_pen;
    MoveL RelTool(pTarget,0,0,-2),vSpeed,z0,tTool\WObj:=wWobj;
    pTarget.trans := [0,12.0,0];
    MoveL pTarget,vSpeed,fine,tTool\WObj:=wWobj;
    Set do_pen;
    pTarget.trans := [2,11.0,0];
    MoveL pTarget,vSpeed,z0,tTool\WObj:=wWobj;
    pTarget.trans := [6,11.0,0];
    MoveL pTarget,vSpeed,z0,tTool\WObj:=wWobj;
    pTarget.trans := [8,12.0,0];
    MoveL pTarget,vSpeed,z0,tTool\WObj:=wWobj;
    pTarget.trans := [9,13.0,0];
    MoveL pTarget,vSpeed,z0,tTool\WObj:=wWobj;
    pTarget.trans := [11,16.0,0];
    MoveL pTarget,vSpeed,fine,tTool\WObj:=wWobj;
    Reset do_pen;
    MoveL RelTool(pTarget,0,0,-2),vSpeed,z0,tTool\WObj:=wWobj;
    wWobj.oframe.trans.x := wWobj.oframe.trans.x + 11;
ENDPROC
  ! Character: t
  PROC char_t()
    VAR robtarget pTarget;
    pTarget := refTarget;
    pTarget.trans := [0,16.0,0];
    MoveL pTarget,vSpeed,fine,tTool\WObj:=wWobj;
    Set do_pen;
    pTarget.trans := [2,19.0,0];
    MoveL pTarget,vSpeed,z0,tTool\WObj:=wWobj;
    pTarget.trans := [4,23.0,0];
    MoveL pTarget,vSpeed,fine,tTool\WObj:=wWobj;
    Reset do_pen;
    MoveL RelTool(pTarget,0,0,-2),vSpeed,z0,tTool\WObj:=wWobj;
    pTarget.trans := [7,32.0,0];
    MoveL pTarget,vSpeed,fine,tTool\WObj:=wWobj;
    Set do_pen;
    pTarget.trans := [1,14.0,0];
    MoveL pTarget,vSpeed,z0,tTool\WObj:=wWobj;
    pTarget.trans := [1,12.0,0];
    MoveL pTarget,vSpeed,z0,tTool\WObj:=wWobj;
    pTarget.trans := [2,11.0,0];
    MoveL pTarget,vSpeed,z0,tTool\WObj:=wWobj;
    pTarget.trans := [4,11.0,0];
    MoveL pTarget,vSpeed,z0,tTool\WObj:=wWobj;
    pTarget.trans := [6,12.0,0];
    MoveL pTarget,vSpeed,z0,tTool\WObj:=wWobj;
    pTarget.trans := [7,13.0,0];
    MoveL pTarget,vSpeed,z0,tTool\WObj:=wWobj;
    pTarget.trans := [9,16.0,0];
    MoveL pTarget,vSpeed,fine,tTool\WObj:=wWobj;
    Reset do_pen;
    MoveL RelTool(pTarget,0,0,-2),vSpeed,z0,tTool\WObj:=wWobj;
    pTarget.trans := [1,24.0,0];
    MoveL pTarget,vSpeed,fine,tTool\WObj:=wWobj;
    Set do_pen;
    pTarget.trans := [8,24.0,0];
    MoveL pTarget,vSpeed,fine,tTool\WObj:=wWobj;
    Reset do_pen;
    MoveL RelTool(pTarget,0,0,-2),vSpeed,z0,tTool\WObj:=wWobj;
    wWobj.oframe.trans.x := wWobj.oframe.trans.x + 9;
ENDPROC
  ! Character: u
  PROC char_u()
    VAR robtarget pTarget;
    pTarget := refTarget;
    pTarget.trans := [0,16.0,0];
    MoveL pTarget,vSpeed,fine,tTool\WObj:=wWobj;
    Set do_pen;
    pTarget.trans := [2,20.0,0];
    MoveL pTarget,vSpeed,z0,tTool\WObj:=wWobj;
    pTarget.trans := [0,14.0,0];
    MoveL pTarget,vSpeed,z0,tTool\WObj:=wWobj;
    pTarget.trans := [0,12.0,0];
    MoveL pTarget,vSpeed,z0,tTool\WObj:=wWobj;
    pTarget.trans := [1,11.0,0];
    MoveL pTarget,vSpeed,z0,tTool\WObj:=wWobj;
    pTarget.trans := [3,11.0,0];
    MoveL pTarget,vSpeed,z0,tTool\WObj:=wWobj;
    pTarget.trans := [5,12.0,0];
    MoveL pTarget,vSpeed,z0,tTool\WObj:=wWobj;
    pTarget.trans := [7,14.0,0];
    MoveL pTarget,vSpeed,z0,tTool\WObj:=wWobj;
    pTarget.trans := [9,17.0,0];
    MoveL pTarget,vSpeed,fine,tTool\WObj:=wWobj;
    Reset do_pen;
    MoveL RelTool(pTarget,0,0,-2),vSpeed,z0,tTool\WObj:=wWobj;
    pTarget.trans := [10,20.0,0];
    MoveL pTarget,vSpeed,fine,tTool\WObj:=wWobj;
    Set do_pen;
    pTarget.trans := [8,14.0,0];
    MoveL pTarget,vSpeed,z0,tTool\WObj:=wWobj;
    pTarget.trans := [8,12.0,0];
    MoveL pTarget,vSpeed,z0,tTool\WObj:=wWobj;
    pTarget.trans := [9,11.0,0];
    MoveL pTarget,vSpeed,z0,tTool\WObj:=wWobj;
    pTarget.trans := [10,11.0,0];
    MoveL pTarget,vSpeed,z0,tTool\WObj:=wWobj;
    pTarget.trans := [12,12.0,0];
    MoveL pTarget,vSpeed,z0,tTool\WObj:=wWobj;
    pTarget.trans := [13,13.0,0];
    MoveL pTarget,vSpeed,z0,tTool\WObj:=wWobj;
    pTarget.trans := [15,16.0,0];
    MoveL pTarget,vSpeed,fine,tTool\WObj:=wWobj;
    Reset do_pen;
    MoveL RelTool(pTarget,0,0,-2),vSpeed,z0,tTool\WObj:=wWobj;
    wWobj.oframe.trans.x := wWobj.oframe.trans.x + 15;
ENDPROC
  ! Character: v
  PROC char_v()
    VAR robtarget pTarget;
    pTarget := refTarget;
    pTarget.trans := [0,16.0,0];
    MoveL pTarget,vSpeed,fine,tTool\WObj:=wWobj;
    Set do_pen;
    pTarget.trans := [2,20.0,0];
    MoveL pTarget,vSpeed,z0,tTool\WObj:=wWobj;
    pTarget.trans := [1,15.0,0];
    MoveL pTarget,vSpeed,z0,tTool\WObj:=wWobj;
    pTarget.trans := [1,12.0,0];
    MoveL pTarget,vSpeed,z0,tTool\WObj:=wWobj;
    pTarget.trans := [2,11.0,0];
    MoveL pTarget,vSpeed,z0,tTool\WObj:=wWobj;
    pTarget.trans := [3,11.0,0];
    MoveL pTarget,vSpeed,z0,tTool\WObj:=wWobj;
    pTarget.trans := [6,12.0,0];
    MoveL pTarget,vSpeed,z0,tTool\WObj:=wWobj;
    pTarget.trans := [8,14.0,0];
    MoveL pTarget,vSpeed,z0,tTool\WObj:=wWobj;
    pTarget.trans := [9,17.0,0];
    MoveL pTarget,vSpeed,z0,tTool\WObj:=wWobj;
    pTarget.trans := [9,20.0,0];
    MoveL pTarget,vSpeed,fine,tTool\WObj:=wWobj;
    Reset do_pen;
    MoveL RelTool(pTarget,0,0,-2),vSpeed,z0,tTool\WObj:=wWobj;
    pTarget.trans := [9,20.0,0];
    MoveL pTarget,vSpeed,fine,tTool\WObj:=wWobj;
    Set do_pen;
    pTarget.trans := [10,16.0,0];
    MoveL pTarget,vSpeed,z0,tTool\WObj:=wWobj;
    pTarget.trans := [11,15.0,0];
    MoveL pTarget,vSpeed,z0,tTool\WObj:=wWobj;
    pTarget.trans := [13,15.0,0];
    MoveL pTarget,vSpeed,z0,tTool\WObj:=wWobj;
    pTarget.trans := [15,16.0,0];
    MoveL pTarget,vSpeed,fine,tTool\WObj:=wWobj;
    Reset do_pen;
    MoveL RelTool(pTarget,0,0,-2),vSpeed,z0,tTool\WObj:=wWobj;
    wWobj.oframe.trans.x := wWobj.oframe.trans.x + 15;
ENDPROC
  ! Character: w
  PROC char_w()
    VAR robtarget pTarget;
    pTarget := refTarget;
    pTarget.trans := [3,20.0,0];
    MoveL pTarget,vSpeed,fine,tTool\WObj:=wWobj;
    Set do_pen;
    pTarget.trans := [1,18.0,0];
    MoveL pTarget,vSpeed,z0,tTool\WObj:=wWobj;
    pTarget.trans := [0,15.0,0];
    MoveL pTarget,vSpeed,z0,tTool\WObj:=wWobj;
    pTarget.trans := [0,13.0,0];
    MoveL pTarget,vSpeed,z0,tTool\WObj:=wWobj;
    pTarget.trans := [1,11.0,0];
    MoveL pTarget,vSpeed,z0,tTool\WObj:=wWobj;
    pTarget.trans := [3,11.0,0];
    MoveL pTarget,vSpeed,z0,tTool\WObj:=wWobj;
    pTarget.trans := [5,12.0,0];
    MoveL pTarget,vSpeed,z0,tTool\WObj:=wWobj;
    pTarget.trans := [7,14.0,0];
    MoveL pTarget,vSpeed,fine,tTool\WObj:=wWobj;
    Reset do_pen;
    MoveL RelTool(pTarget,0,0,-2),vSpeed,z0,tTool\WObj:=wWobj;
    pTarget.trans := [9,20.0,0];
    MoveL pTarget,vSpeed,fine,tTool\WObj:=wWobj;
    Set do_pen;
    pTarget.trans := [7,14.0,0];
    MoveL pTarget,vSpeed,z0,tTool\WObj:=wWobj;
    pTarget.trans := [7,12.0,0];
    MoveL pTarget,vSpeed,z0,tTool\WObj:=wWobj;
    pTarget.trans := [8,11.0,0];
    MoveL pTarget,vSpeed,z0,tTool\WObj:=wWobj;
    pTarget.trans := [10,11.0,0];
    MoveL pTarget,vSpeed,z0,tTool\WObj:=wWobj;
    pTarget.trans := [12,12.0,0];
    MoveL pTarget,vSpeed,z0,tTool\WObj:=wWobj;
    pTarget.trans := [14,14.0,0];
    MoveL pTarget,vSpeed,z0,tTool\WObj:=wWobj;
    pTarget.trans := [15,17.0,0];
    MoveL pTarget,vSpeed,z0,tTool\WObj:=wWobj;
    pTarget.trans := [15,20.0,0];
    MoveL pTarget,vSpeed,fine,tTool\WObj:=wWobj;
    Reset do_pen;
    MoveL RelTool(pTarget,0,0,-2),vSpeed,z0,tTool\WObj:=wWobj;
    pTarget.trans := [15,20.0,0];
    MoveL pTarget,vSpeed,fine,tTool\WObj:=wWobj;
    Set do_pen;
    pTarget.trans := [16,16.0,0];
    MoveL pTarget,vSpeed,z0,tTool\WObj:=wWobj;
    pTarget.trans := [17,15.0,0];
    MoveL pTarget,vSpeed,z0,tTool\WObj:=wWobj;
    pTarget.trans := [19,15.0,0];
    MoveL pTarget,vSpeed,z0,tTool\WObj:=wWobj;
    pTarget.trans := [21,16.0,0];
    MoveL pTarget,vSpeed,fine,tTool\WObj:=wWobj;
    Reset do_pen;
    MoveL RelTool(pTarget,0,0,-2),vSpeed,z0,tTool\WObj:=wWobj;
    wWobj.oframe.trans.x := wWobj.oframe.trans.x + 21;
ENDPROC
  ! Character: x
  PROC char_x()
    VAR robtarget pTarget;
    pTarget := refTarget;
    pTarget.trans := [0,16.0,0];
    MoveL pTarget,vSpeed,fine,tTool\WObj:=wWobj;
    Set do_pen;
    pTarget.trans := [2,19.0,0];
    MoveL pTarget,vSpeed,z0,tTool\WObj:=wWobj;
    pTarget.trans := [4,20.0,0];
    MoveL pTarget,vSpeed,z0,tTool\WObj:=wWobj;
    pTarget.trans := [6,20.0,0];
    MoveL pTarget,vSpeed,z0,tTool\WObj:=wWobj;
    pTarget.trans := [7,19.0,0];
    MoveL pTarget,vSpeed,z0,tTool\WObj:=wWobj;
    pTarget.trans := [7,12.0,0];
    MoveL pTarget,vSpeed,z0,tTool\WObj:=wWobj;
    pTarget.trans := [8,11.0,0];
    MoveL pTarget,vSpeed,z0,tTool\WObj:=wWobj;
    pTarget.trans := [11,11.0,0];
    MoveL pTarget,vSpeed,z0,tTool\WObj:=wWobj;
    pTarget.trans := [14,13.0,0];
    MoveL pTarget,vSpeed,z0,tTool\WObj:=wWobj;
    pTarget.trans := [16,16.0,0];
    MoveL pTarget,vSpeed,fine,tTool\WObj:=wWobj;
    Reset do_pen;
    MoveL RelTool(pTarget,0,0,-2),vSpeed,z0,tTool\WObj:=wWobj;
    pTarget.trans := [13,19.0,0];
    MoveL pTarget,vSpeed,fine,tTool\WObj:=wWobj;
    Set do_pen;
    pTarget.trans := [12,20.0,0];
    MoveL pTarget,vSpeed,z0,tTool\WObj:=wWobj;
    pTarget.trans := [10,20.0,0];
    MoveL pTarget,vSpeed,z0,tTool\WObj:=wWobj;
    pTarget.trans := [9,19.0,0];
    MoveL pTarget,vSpeed,z0,tTool\WObj:=wWobj;
    pTarget.trans := [5,12.0,0];
    MoveL pTarget,vSpeed,z0,tTool\WObj:=wWobj;
    pTarget.trans := [4,11.0,0];
    MoveL pTarget,vSpeed,z0,tTool\WObj:=wWobj;
    pTarget.trans := [2,11.0,0];
    MoveL pTarget,vSpeed,z0,tTool\WObj:=wWobj;
    pTarget.trans := [1,12.0,0];
    MoveL pTarget,vSpeed,fine,tTool\WObj:=wWobj;
    Reset do_pen;
    MoveL RelTool(pTarget,0,0,-2),vSpeed,z0,tTool\WObj:=wWobj;
    wWobj.oframe.trans.x := wWobj.oframe.trans.x + 16;
ENDPROC
  ! Character: y
  PROC char_y()
    VAR robtarget pTarget;
    pTarget := refTarget;
    pTarget.trans := [0,16.0,0];
    MoveL pTarget,vSpeed,fine,tTool\WObj:=wWobj;
    Set do_pen;
    pTarget.trans := [2,20.0,0];
    MoveL pTarget,vSpeed,z0,tTool\WObj:=wWobj;
    pTarget.trans := [0,14.0,0];
    MoveL pTarget,vSpeed,z0,tTool\WObj:=wWobj;
    pTarget.trans := [0,12.0,0];
    MoveL pTarget,vSpeed,z0,tTool\WObj:=wWobj;
    pTarget.trans := [1,11.0,0];
    MoveL pTarget,vSpeed,z0,tTool\WObj:=wWobj;
    pTarget.trans := [3,11.0,0];
    MoveL pTarget,vSpeed,z0,tTool\WObj:=wWobj;
    pTarget.trans := [5,12.0,0];
    MoveL pTarget,vSpeed,z0,tTool\WObj:=wWobj;
    pTarget.trans := [7,14.0,0];
    MoveL pTarget,vSpeed,z0,tTool\WObj:=wWobj;
    pTarget.trans := [9,17.0,0];
    MoveL pTarget,vSpeed,fine,tTool\WObj:=wWobj;
    Reset do_pen;
    MoveL RelTool(pTarget,0,0,-2),vSpeed,z0,tTool\WObj:=wWobj;
    pTarget.trans := [10,20.0,0];
    MoveL pTarget,vSpeed,fine,tTool\WObj:=wWobj;
    Set do_pen;
    pTarget.trans := [4,2.0,0];
    MoveL pTarget,vSpeed,z0,tTool\WObj:=wWobj;
    pTarget.trans := [3,0.0,0];
    MoveL pTarget,vSpeed,z0,tTool\WObj:=wWobj;
    pTarget.trans := [1,-1.0,0];
    MoveL pTarget,vSpeed,z0,tTool\WObj:=wWobj;
    pTarget.trans := [0,0.0,0];
    MoveL pTarget,vSpeed,z0,tTool\WObj:=wWobj;
    pTarget.trans := [0,2.0,0];
    MoveL pTarget,vSpeed,z0,tTool\WObj:=wWobj;
    pTarget.trans := [1,5.0,0];
    MoveL pTarget,vSpeed,z0,tTool\WObj:=wWobj;
    pTarget.trans := [4,8.0,0];
    MoveL pTarget,vSpeed,z0,tTool\WObj:=wWobj;
    pTarget.trans := [7,10.0,0];
    MoveL pTarget,vSpeed,z0,tTool\WObj:=wWobj;
    pTarget.trans := [9,11.0,0];
    MoveL pTarget,vSpeed,z0,tTool\WObj:=wWobj;
    pTarget.trans := [12,13.0,0];
    MoveL pTarget,vSpeed,z0,tTool\WObj:=wWobj;
    pTarget.trans := [15,16.0,0];
    MoveL pTarget,vSpeed,fine,tTool\WObj:=wWobj;
    Reset do_pen;
    MoveL RelTool(pTarget,0,0,-2),vSpeed,z0,tTool\WObj:=wWobj;
    wWobj.oframe.trans.x := wWobj.oframe.trans.x + 15;
ENDPROC
  ! Character: z
  PROC char_z()
    VAR robtarget pTarget;
    pTarget := refTarget;
    pTarget.trans := [0,16.0,0];
    MoveL pTarget,vSpeed,fine,tTool\WObj:=wWobj;
    Set do_pen;
    pTarget.trans := [2,19.0,0];
    MoveL pTarget,vSpeed,z0,tTool\WObj:=wWobj;
    pTarget.trans := [4,20.0,0];
    MoveL pTarget,vSpeed,z0,tTool\WObj:=wWobj;
    pTarget.trans := [6,20.0,0];
    MoveL pTarget,vSpeed,z0,tTool\WObj:=wWobj;
    pTarget.trans := [8,18.0,0];
    MoveL pTarget,vSpeed,z0,tTool\WObj:=wWobj;
    pTarget.trans := [8,16.0,0];
    MoveL pTarget,vSpeed,z0,tTool\WObj:=wWobj;
    pTarget.trans := [7,14.0,0];
    MoveL pTarget,vSpeed,z0,tTool\WObj:=wWobj;
    pTarget.trans := [5,12.0,0];
    MoveL pTarget,vSpeed,z0,tTool\WObj:=wWobj;
    pTarget.trans := [2,11.0,0];
    MoveL pTarget,vSpeed,z0,tTool\WObj:=wWobj;
    pTarget.trans := [4,10.0,0];
    MoveL pTarget,vSpeed,z0,tTool\WObj:=wWobj;
    pTarget.trans := [5,8.0,0];
    MoveL pTarget,vSpeed,z0,tTool\WObj:=wWobj;
    pTarget.trans := [5,5.0,0];
    MoveL pTarget,vSpeed,z0,tTool\WObj:=wWobj;
    pTarget.trans := [4,2.0,0];
    MoveL pTarget,vSpeed,z0,tTool\WObj:=wWobj;
    pTarget.trans := [3,0.0,0];
    MoveL pTarget,vSpeed,z0,tTool\WObj:=wWobj;
    pTarget.trans := [1,-1.0,0];
    MoveL pTarget,vSpeed,z0,tTool\WObj:=wWobj;
    pTarget.trans := [0,0.0,0];
    MoveL pTarget,vSpeed,z0,tTool\WObj:=wWobj;
    pTarget.trans := [0,2.0,0];
    MoveL pTarget,vSpeed,z0,tTool\WObj:=wWobj;
    pTarget.trans := [1,5.0,0];
    MoveL pTarget,vSpeed,z0,tTool\WObj:=wWobj;
    pTarget.trans := [4,8.0,0];
    MoveL pTarget,vSpeed,z0,tTool\WObj:=wWobj;
    pTarget.trans := [7,10.0,0];
    MoveL pTarget,vSpeed,z0,tTool\WObj:=wWobj;
    pTarget.trans := [11,13.0,0];
    MoveL pTarget,vSpeed,z0,tTool\WObj:=wWobj;
    pTarget.trans := [14,16.0,0];
    MoveL pTarget,vSpeed,fine,tTool\WObj:=wWobj;
    Reset do_pen;
    MoveL RelTool(pTarget,0,0,-2),vSpeed,z0,tTool\WObj:=wWobj;
    wWobj.oframe.trans.x := wWobj.oframe.trans.x + 14;
ENDPROC
  ! Character: A
  PROC char_upperA()
    VAR robtarget pTarget;
    pTarget := refTarget;
    pTarget.trans := [0,11.0,0];
    MoveL pTarget,vSpeed,fine,tTool\WObj:=wWobj;
    Set do_pen;
    pTarget.trans := [2,12.0,0];
    MoveL pTarget,vSpeed,z0,tTool\WObj:=wWobj;
    pTarget.trans := [5,15.0,0];
    MoveL pTarget,vSpeed,z0,tTool\WObj:=wWobj;
    pTarget.trans := [8,19.0,0];
    MoveL pTarget,vSpeed,z0,tTool\WObj:=wWobj;
    pTarget.trans := [12,26.0,0];
    MoveL pTarget,vSpeed,z0,tTool\WObj:=wWobj;
    pTarget.trans := [15,32.0,0];
    MoveL pTarget,vSpeed,z0,tTool\WObj:=wWobj;
    pTarget.trans := [15,11.0,0];
    MoveL pTarget,vSpeed,z0,tTool\WObj:=wWobj;
    pTarget.trans := [14,14.0,0];
    MoveL pTarget,vSpeed,z0,tTool\WObj:=wWobj;
    pTarget.trans := [12,17.0,0];
    MoveL pTarget,vSpeed,z0,tTool\WObj:=wWobj;
    pTarget.trans := [10,19.0,0];
    MoveL pTarget,vSpeed,z0,tTool\WObj:=wWobj;
    pTarget.trans := [7,21.0,0];
    MoveL pTarget,vSpeed,z0,tTool\WObj:=wWobj;
    pTarget.trans := [5,21.0,0];
    MoveL pTarget,vSpeed,z0,tTool\WObj:=wWobj;
    pTarget.trans := [4,20.0,0];
    MoveL pTarget,vSpeed,z0,tTool\WObj:=wWobj;
    pTarget.trans := [4,18.0,0];
    MoveL pTarget,vSpeed,z0,tTool\WObj:=wWobj;
    pTarget.trans := [5,16.0,0];
    MoveL pTarget,vSpeed,z0,tTool\WObj:=wWobj;
    pTarget.trans := [7,14.0,0];
    MoveL pTarget,vSpeed,z0,tTool\WObj:=wWobj;
    pTarget.trans := [10,12.0,0];
    MoveL pTarget,vSpeed,z0,tTool\WObj:=wWobj;
    pTarget.trans := [13,11.0,0];
    MoveL pTarget,vSpeed,z0,tTool\WObj:=wWobj;
    pTarget.trans := [18,11.0,0];
    MoveL pTarget,vSpeed,fine,tTool\WObj:=wWobj;
    Reset do_pen;
    MoveL RelTool(pTarget,0,0,-2),vSpeed,z0,tTool\WObj:=wWobj;
    wWobj.oframe.trans.x := wWobj.oframe.trans.x + 18;
ENDPROC
  ! Character: B
  PROC char_upperB()
    VAR robtarget pTarget;
    pTarget := refTarget;
    pTarget.trans := [13,30.0,0];
    MoveL pTarget,vSpeed,fine,tTool\WObj:=wWobj;
    Set do_pen;
    pTarget.trans := [14,29.0,0];
    MoveL pTarget,vSpeed,z0,tTool\WObj:=wWobj;
    pTarget.trans := [14,26.0,0];
    MoveL pTarget,vSpeed,z0,tTool\WObj:=wWobj;
    pTarget.trans := [13,22.0,0];
    MoveL pTarget,vSpeed,z0,tTool\WObj:=wWobj;
    pTarget.trans := [12,19.0,0];
    MoveL pTarget,vSpeed,z0,tTool\WObj:=wWobj;
    pTarget.trans := [11,17.0,0];
    MoveL pTarget,vSpeed,z0,tTool\WObj:=wWobj;
    pTarget.trans := [9,14.0,0];
    MoveL pTarget,vSpeed,z0,tTool\WObj:=wWobj;
    pTarget.trans := [7,12.0,0];
    MoveL pTarget,vSpeed,z0,tTool\WObj:=wWobj;
    pTarget.trans := [5,11.0,0];
    MoveL pTarget,vSpeed,z0,tTool\WObj:=wWobj;
    pTarget.trans := [4,11.0,0];
    MoveL pTarget,vSpeed,z0,tTool\WObj:=wWobj;
    pTarget.trans := [3,12.0,0];
    MoveL pTarget,vSpeed,z0,tTool\WObj:=wWobj;
    pTarget.trans := [3,15.0,0];
    MoveL pTarget,vSpeed,z0,tTool\WObj:=wWobj;
    pTarget.trans := [4,20.0,0];
    MoveL pTarget,vSpeed,z0,tTool\WObj:=wWobj;
    pTarget.trans := [5,23.0,0];
    MoveL pTarget,vSpeed,z0,tTool\WObj:=wWobj;
    pTarget.trans := [6,25.0,0];
    MoveL pTarget,vSpeed,z0,tTool\WObj:=wWobj;
    pTarget.trans := [8,28.0,0];
    MoveL pTarget,vSpeed,z0,tTool\WObj:=wWobj;
    pTarget.trans := [10,30.0,0];
    MoveL pTarget,vSpeed,z0,tTool\WObj:=wWobj;
    pTarget.trans := [12,31.0,0];
    MoveL pTarget,vSpeed,z0,tTool\WObj:=wWobj;
    pTarget.trans := [15,32.0,0];
    MoveL pTarget,vSpeed,z0,tTool\WObj:=wWobj;
    pTarget.trans := [18,32.0,0];
    MoveL pTarget,vSpeed,z0,tTool\WObj:=wWobj;
    pTarget.trans := [20,31.0,0];
    MoveL pTarget,vSpeed,z0,tTool\WObj:=wWobj;
    pTarget.trans := [21,29.0,0];
    MoveL pTarget,vSpeed,z0,tTool\WObj:=wWobj;
    pTarget.trans := [21,27.0,0];
    MoveL pTarget,vSpeed,z0,tTool\WObj:=wWobj;
    pTarget.trans := [20,25.0,0];
    MoveL pTarget,vSpeed,z0,tTool\WObj:=wWobj;
    pTarget.trans := [19,24.0,0];
    MoveL pTarget,vSpeed,z0,tTool\WObj:=wWobj;
    pTarget.trans := [17,23.0,0];
    MoveL pTarget,vSpeed,z0,tTool\WObj:=wWobj;
    pTarget.trans := [14,22.0,0];
    MoveL pTarget,vSpeed,fine,tTool\WObj:=wWobj;
    Reset do_pen;
    MoveL RelTool(pTarget,0,0,-2),vSpeed,z0,tTool\WObj:=wWobj;
    pTarget.trans := [13,22.0,0];
    MoveL pTarget,vSpeed,fine,tTool\WObj:=wWobj;
    Set do_pen;
    pTarget.trans := [14,22.0,0];
    MoveL pTarget,vSpeed,z0,tTool\WObj:=wWobj;
    pTarget.trans := [17,21.0,0];
    MoveL pTarget,vSpeed,z0,tTool\WObj:=wWobj;
    pTarget.trans := [18,20.0,0];
    MoveL pTarget,vSpeed,z0,tTool\WObj:=wWobj;
    pTarget.trans := [19,18.0,0];
    MoveL pTarget,vSpeed,z0,tTool\WObj:=wWobj;
    pTarget.trans := [19,15.0,0];
    MoveL pTarget,vSpeed,z0,tTool\WObj:=wWobj;
    pTarget.trans := [18,13.0,0];
    MoveL pTarget,vSpeed,z0,tTool\WObj:=wWobj;
    pTarget.trans := [17,12.0,0];
    MoveL pTarget,vSpeed,z0,tTool\WObj:=wWobj;
    pTarget.trans := [15,11.0,0];
    MoveL pTarget,vSpeed,z0,tTool\WObj:=wWobj;
    pTarget.trans := [12,11.0,0];
    MoveL pTarget,vSpeed,z0,tTool\WObj:=wWobj;
    pTarget.trans := [10,12.0,0];
    MoveL pTarget,vSpeed,z0,tTool\WObj:=wWobj;
    pTarget.trans := [9,14.0,0];
    MoveL pTarget,vSpeed,fine,tTool\WObj:=wWobj;
    Reset do_pen;
    MoveL RelTool(pTarget,0,0,-2),vSpeed,z0,tTool\WObj:=wWobj;
    wWobj.oframe.trans.x := wWobj.oframe.trans.x + 18;
ENDPROC
  ! Character: C
  PROC char_upperC()
    VAR robtarget pTarget;
    pTarget := refTarget;
    pTarget.trans := [12,26.0,0];
    MoveL pTarget,vSpeed,fine,tTool\WObj:=wWobj;
    Set do_pen;
    pTarget.trans := [12,25.0,0];
    MoveL pTarget,vSpeed,z0,tTool\WObj:=wWobj;
    pTarget.trans := [13,24.0,0];
    MoveL pTarget,vSpeed,z0,tTool\WObj:=wWobj;
    pTarget.trans := [15,24.0,0];
    MoveL pTarget,vSpeed,z0,tTool\WObj:=wWobj;
    pTarget.trans := [17,25.0,0];
    MoveL pTarget,vSpeed,z0,tTool\WObj:=wWobj;
    pTarget.trans := [18,27.0,0];
    MoveL pTarget,vSpeed,z0,tTool\WObj:=wWobj;
    pTarget.trans := [18,29.0,0];
    MoveL pTarget,vSpeed,z0,tTool\WObj:=wWobj;
    pTarget.trans := [17,31.0,0];
    MoveL pTarget,vSpeed,z0,tTool\WObj:=wWobj;
    pTarget.trans := [15,32.0,0];
    MoveL pTarget,vSpeed,z0,tTool\WObj:=wWobj;
    pTarget.trans := [12,32.0,0];
    MoveL pTarget,vSpeed,z0,tTool\WObj:=wWobj;
    pTarget.trans := [9,31.0,0];
    MoveL pTarget,vSpeed,z0,tTool\WObj:=wWobj;
    pTarget.trans := [7,29.0,0];
    MoveL pTarget,vSpeed,z0,tTool\WObj:=wWobj;
    pTarget.trans := [5,26.0,0];
    MoveL pTarget,vSpeed,z0,tTool\WObj:=wWobj;
    pTarget.trans := [4,24.0,0];
    MoveL pTarget,vSpeed,z0,tTool\WObj:=wWobj;
    pTarget.trans := [3,20.0,0];
    MoveL pTarget,vSpeed,z0,tTool\WObj:=wWobj;
    pTarget.trans := [3,16.0,0];
    MoveL pTarget,vSpeed,z0,tTool\WObj:=wWobj;
    pTarget.trans := [4,13.0,0];
    MoveL pTarget,vSpeed,z0,tTool\WObj:=wWobj;
    pTarget.trans := [5,12.0,0];
    MoveL pTarget,vSpeed,z0,tTool\WObj:=wWobj;
    pTarget.trans := [7,11.0,0];
    MoveL pTarget,vSpeed,z0,tTool\WObj:=wWobj;
    pTarget.trans := [9,11.0,0];
    MoveL pTarget,vSpeed,z0,tTool\WObj:=wWobj;
    pTarget.trans := [12,12.0,0];
    MoveL pTarget,vSpeed,z0,tTool\WObj:=wWobj;
    pTarget.trans := [14,14.0,0];
    MoveL pTarget,vSpeed,z0,tTool\WObj:=wWobj;
    pTarget.trans := [15,16.0,0];
    MoveL pTarget,vSpeed,fine,tTool\WObj:=wWobj;
    Reset do_pen;
    MoveL RelTool(pTarget,0,0,-2),vSpeed,z0,tTool\WObj:=wWobj;
    wWobj.oframe.trans.x := wWobj.oframe.trans.x + 15;
ENDPROC
  ! Character: D
  PROC char_upperD()
    VAR robtarget pTarget;
    pTarget := refTarget;
    pTarget.trans := [13,32.0,0];
    MoveL pTarget,vSpeed,fine,tTool\WObj:=wWobj;
    Set do_pen;
    pTarget.trans := [11,31.0,0];
    MoveL pTarget,vSpeed,z0,tTool\WObj:=wWobj;
    pTarget.trans := [10,29.0,0];
    MoveL pTarget,vSpeed,z0,tTool\WObj:=wWobj;
    pTarget.trans := [9,25.0,0];
    MoveL pTarget,vSpeed,z0,tTool\WObj:=wWobj;
    pTarget.trans := [8,19.0,0];
    MoveL pTarget,vSpeed,z0,tTool\WObj:=wWobj;
    pTarget.trans := [7,16.0,0];
    MoveL pTarget,vSpeed,z0,tTool\WObj:=wWobj;
    pTarget.trans := [6,14.0,0];
    MoveL pTarget,vSpeed,z0,tTool\WObj:=wWobj;
    pTarget.trans := [4,12.0,0];
    MoveL pTarget,vSpeed,z0,tTool\WObj:=wWobj;
    pTarget.trans := [2,11.0,0];
    MoveL pTarget,vSpeed,z0,tTool\WObj:=wWobj;
    pTarget.trans := [0,11.0,0];
    MoveL pTarget,vSpeed,z0,tTool\WObj:=wWobj;
    pTarget.trans := [-1,12.0,0];
    MoveL pTarget,vSpeed,z0,tTool\WObj:=wWobj;
    pTarget.trans := [-1,14.0,0];
    MoveL pTarget,vSpeed,z0,tTool\WObj:=wWobj;
    pTarget.trans := [0,15.0,0];
    MoveL pTarget,vSpeed,z0,tTool\WObj:=wWobj;
    pTarget.trans := [2,15.0,0];
    MoveL pTarget,vSpeed,z0,tTool\WObj:=wWobj;
    pTarget.trans := [4,14.0,0];
    MoveL pTarget,vSpeed,z0,tTool\WObj:=wWobj;
    pTarget.trans := [6,12.0,0];
    MoveL pTarget,vSpeed,z0,tTool\WObj:=wWobj;
    pTarget.trans := [9,11.0,0];
    MoveL pTarget,vSpeed,z0,tTool\WObj:=wWobj;
    pTarget.trans := [12,11.0,0];
    MoveL pTarget,vSpeed,z0,tTool\WObj:=wWobj;
    pTarget.trans := [15,12.0,0];
    MoveL pTarget,vSpeed,z0,tTool\WObj:=wWobj;
    pTarget.trans := [17,14.0,0];
    MoveL pTarget,vSpeed,z0,tTool\WObj:=wWobj;
    pTarget.trans := [19,18.0,0];
    MoveL pTarget,vSpeed,z0,tTool\WObj:=wWobj;
    pTarget.trans := [20,23.0,0];
    MoveL pTarget,vSpeed,z0,tTool\WObj:=wWobj;
    pTarget.trans := [20,27.0,0];
    MoveL pTarget,vSpeed,z0,tTool\WObj:=wWobj;
    pTarget.trans := [19,30.0,0];
    MoveL pTarget,vSpeed,z0,tTool\WObj:=wWobj;
    pTarget.trans := [18,31.0,0];
    MoveL pTarget,vSpeed,z0,tTool\WObj:=wWobj;
    pTarget.trans := [16,32.0,0];
    MoveL pTarget,vSpeed,z0,tTool\WObj:=wWobj;
    pTarget.trans := [13,32.0,0];
    MoveL pTarget,vSpeed,z0,tTool\WObj:=wWobj;
    pTarget.trans := [11,30.0,0];
    MoveL pTarget,vSpeed,z0,tTool\WObj:=wWobj;
    pTarget.trans := [11,28.0,0];
    MoveL pTarget,vSpeed,z0,tTool\WObj:=wWobj;
    pTarget.trans := [12,25.0,0];
    MoveL pTarget,vSpeed,z0,tTool\WObj:=wWobj;
    pTarget.trans := [14,22.0,0];
    MoveL pTarget,vSpeed,z0,tTool\WObj:=wWobj;
    pTarget.trans := [16,20.0,0];
    MoveL pTarget,vSpeed,z0,tTool\WObj:=wWobj;
    pTarget.trans := [19,18.0,0];
    MoveL pTarget,vSpeed,z0,tTool\WObj:=wWobj;
    pTarget.trans := [21,17.0,0];
    MoveL pTarget,vSpeed,fine,tTool\WObj:=wWobj;
    Reset do_pen;
    MoveL RelTool(pTarget,0,0,-2),vSpeed,z0,tTool\WObj:=wWobj;
    wWobj.oframe.trans.x := wWobj.oframe.trans.x + 22;
ENDPROC
  ! Character: E
  PROC char_upperE()
    VAR robtarget pTarget;
    pTarget := refTarget;
    pTarget.trans := [14,28.0,0];
    MoveL pTarget,vSpeed,fine,tTool\WObj:=wWobj;
    Set do_pen;
    pTarget.trans := [14,27.0,0];
    MoveL pTarget,vSpeed,z0,tTool\WObj:=wWobj;
    pTarget.trans := [15,26.0,0];
    MoveL pTarget,vSpeed,z0,tTool\WObj:=wWobj;
    pTarget.trans := [17,26.0,0];
    MoveL pTarget,vSpeed,z0,tTool\WObj:=wWobj;
    pTarget.trans := [18,27.0,0];
    MoveL pTarget,vSpeed,z0,tTool\WObj:=wWobj;
    pTarget.trans := [18,29.0,0];
    MoveL pTarget,vSpeed,z0,tTool\WObj:=wWobj;
    pTarget.trans := [17,31.0,0];
    MoveL pTarget,vSpeed,z0,tTool\WObj:=wWobj;
    pTarget.trans := [14,32.0,0];
    MoveL pTarget,vSpeed,z0,tTool\WObj:=wWobj;
    pTarget.trans := [10,32.0,0];
    MoveL pTarget,vSpeed,z0,tTool\WObj:=wWobj;
    pTarget.trans := [7,31.0,0];
    MoveL pTarget,vSpeed,z0,tTool\WObj:=wWobj;
    pTarget.trans := [6,29.0,0];
    MoveL pTarget,vSpeed,z0,tTool\WObj:=wWobj;
    pTarget.trans := [6,26.0,0];
    MoveL pTarget,vSpeed,z0,tTool\WObj:=wWobj;
    pTarget.trans := [7,24.0,0];
    MoveL pTarget,vSpeed,z0,tTool\WObj:=wWobj;
    pTarget.trans := [8,23.0,0];
    MoveL pTarget,vSpeed,z0,tTool\WObj:=wWobj;
    pTarget.trans := [11,22.0,0];
    MoveL pTarget,vSpeed,z0,tTool\WObj:=wWobj;
    pTarget.trans := [8,22.0,0];
    MoveL pTarget,vSpeed,z0,tTool\WObj:=wWobj;
    pTarget.trans := [5,21.0,0];
    MoveL pTarget,vSpeed,z0,tTool\WObj:=wWobj;
    pTarget.trans := [4,20.0,0];
    MoveL pTarget,vSpeed,z0,tTool\WObj:=wWobj;
    pTarget.trans := [3,18.0,0];
    MoveL pTarget,vSpeed,z0,tTool\WObj:=wWobj;
    pTarget.trans := [3,15.0,0];
    MoveL pTarget,vSpeed,z0,tTool\WObj:=wWobj;
    pTarget.trans := [4,13.0,0];
    MoveL pTarget,vSpeed,z0,tTool\WObj:=wWobj;
    pTarget.trans := [5,12.0,0];
    MoveL pTarget,vSpeed,z0,tTool\WObj:=wWobj;
    pTarget.trans := [8,11.0,0];
    MoveL pTarget,vSpeed,z0,tTool\WObj:=wWobj;
    pTarget.trans := [11,11.0,0];
    MoveL pTarget,vSpeed,z0,tTool\WObj:=wWobj;
    pTarget.trans := [14,12.0,0];
    MoveL pTarget,vSpeed,z0,tTool\WObj:=wWobj;
    pTarget.trans := [16,14.0,0];
    MoveL pTarget,vSpeed,z0,tTool\WObj:=wWobj;
    pTarget.trans := [17,16.0,0];
    MoveL pTarget,vSpeed,fine,tTool\WObj:=wWobj;
    Reset do_pen;
    MoveL RelTool(pTarget,0,0,-2),vSpeed,z0,tTool\WObj:=wWobj;
    wWobj.oframe.trans.x := wWobj.oframe.trans.x + 15;
ENDPROC
  ! Character: F
  PROC char_upperF()
    VAR robtarget pTarget;
    pTarget := refTarget;
    pTarget.trans := [10,26.0,0];
    MoveL pTarget,vSpeed,fine,tTool\WObj:=wWobj;
    Set do_pen;
    pTarget.trans := [8,26.0,0];
    MoveL pTarget,vSpeed,z0,tTool\WObj:=wWobj;
    pTarget.trans := [6,27.0,0];
    MoveL pTarget,vSpeed,z0,tTool\WObj:=wWobj;
    pTarget.trans := [5,29.0,0];
    MoveL pTarget,vSpeed,z0,tTool\WObj:=wWobj;
    pTarget.trans := [6,31.0,0];
    MoveL pTarget,vSpeed,z0,tTool\WObj:=wWobj;
    pTarget.trans := [9,32.0,0];
    MoveL pTarget,vSpeed,z0,tTool\WObj:=wWobj;
    pTarget.trans := [12,32.0,0];
    MoveL pTarget,vSpeed,z0,tTool\WObj:=wWobj;
    pTarget.trans := [16,31.0,0];
    MoveL pTarget,vSpeed,z0,tTool\WObj:=wWobj;
    pTarget.trans := [19,31.0,0];
    MoveL pTarget,vSpeed,z0,tTool\WObj:=wWobj;
    pTarget.trans := [21,32.0,0];
    MoveL pTarget,vSpeed,fine,tTool\WObj:=wWobj;
    Reset do_pen;
    MoveL RelTool(pTarget,0,0,-2),vSpeed,z0,tTool\WObj:=wWobj;
    pTarget.trans := [16,31.0,0];
    MoveL pTarget,vSpeed,fine,tTool\WObj:=wWobj;
    Set do_pen;
    pTarget.trans := [14,24.0,0];
    MoveL pTarget,vSpeed,z0,tTool\WObj:=wWobj;
    pTarget.trans := [12,18.0,0];
    MoveL pTarget,vSpeed,z0,tTool\WObj:=wWobj;
    pTarget.trans := [10,14.0,0];
    MoveL pTarget,vSpeed,z0,tTool\WObj:=wWobj;
    pTarget.trans := [8,12.0,0];
    MoveL pTarget,vSpeed,z0,tTool\WObj:=wWobj;
    pTarget.trans := [6,11.0,0];
    MoveL pTarget,vSpeed,z0,tTool\WObj:=wWobj;
    pTarget.trans := [4,11.0,0];
    MoveL pTarget,vSpeed,z0,tTool\WObj:=wWobj;
    pTarget.trans := [2,12.0,0];
    MoveL pTarget,vSpeed,z0,tTool\WObj:=wWobj;
    pTarget.trans := [1,14.0,0];
    MoveL pTarget,vSpeed,z0,tTool\WObj:=wWobj;
    pTarget.trans := [1,16.0,0];
    MoveL pTarget,vSpeed,z0,tTool\WObj:=wWobj;
    pTarget.trans := [2,17.0,0];
    MoveL pTarget,vSpeed,z0,tTool\WObj:=wWobj;
    pTarget.trans := [4,17.0,0];
    MoveL pTarget,vSpeed,z0,tTool\WObj:=wWobj;
    pTarget.trans := [6,16.0,0];
    MoveL pTarget,vSpeed,fine,tTool\WObj:=wWobj;
    Reset do_pen;
    MoveL RelTool(pTarget,0,0,-2),vSpeed,z0,tTool\WObj:=wWobj;
    pTarget.trans := [9,22.0,0];
    MoveL pTarget,vSpeed,fine,tTool\WObj:=wWobj;
    Set do_pen;
    pTarget.trans := [18,22.0,0];
    MoveL pTarget,vSpeed,fine,tTool\WObj:=wWobj;
    Reset do_pen;
    MoveL RelTool(pTarget,0,0,-2),vSpeed,z0,tTool\WObj:=wWobj;
    wWobj.oframe.trans.x := wWobj.oframe.trans.x + 20;
ENDPROC
  ! Character: G
  PROC char_upperG()
    VAR robtarget pTarget;
    pTarget := refTarget;
    pTarget.trans := [0,11.0,0];
    MoveL pTarget,vSpeed,fine,tTool\WObj:=wWobj;
    Set do_pen;
    pTarget.trans := [2,12.0,0];
    MoveL pTarget,vSpeed,z0,tTool\WObj:=wWobj;
    pTarget.trans := [6,16.0,0];
    MoveL pTarget,vSpeed,z0,tTool\WObj:=wWobj;
    pTarget.trans := [9,21.0,0];
    MoveL pTarget,vSpeed,z0,tTool\WObj:=wWobj;
    pTarget.trans := [10,24.0,0];
    MoveL pTarget,vSpeed,z0,tTool\WObj:=wWobj;
    pTarget.trans := [11,28.0,0];
    MoveL pTarget,vSpeed,z0,tTool\WObj:=wWobj;
    pTarget.trans := [11,31.0,0];
    MoveL pTarget,vSpeed,z0,tTool\WObj:=wWobj;
    pTarget.trans := [10,32.0,0];
    MoveL pTarget,vSpeed,z0,tTool\WObj:=wWobj;
    pTarget.trans := [9,32.0,0];
    MoveL pTarget,vSpeed,z0,tTool\WObj:=wWobj;
    pTarget.trans := [8,31.0,0];
    MoveL pTarget,vSpeed,z0,tTool\WObj:=wWobj;
    pTarget.trans := [7,29.0,0];
    MoveL pTarget,vSpeed,z0,tTool\WObj:=wWobj;
    pTarget.trans := [7,26.0,0];
    MoveL pTarget,vSpeed,z0,tTool\WObj:=wWobj;
    pTarget.trans := [8,24.0,0];
    MoveL pTarget,vSpeed,z0,tTool\WObj:=wWobj;
    pTarget.trans := [10,23.0,0];
    MoveL pTarget,vSpeed,z0,tTool\WObj:=wWobj;
    pTarget.trans := [14,23.0,0];
    MoveL pTarget,vSpeed,z0,tTool\WObj:=wWobj;
    pTarget.trans := [17,24.0,0];
    MoveL pTarget,vSpeed,z0,tTool\WObj:=wWobj;
    pTarget.trans := [18,25.0,0];
    MoveL pTarget,vSpeed,z0,tTool\WObj:=wWobj;
    pTarget.trans := [19,27.0,0];
    MoveL pTarget,vSpeed,z0,tTool\WObj:=wWobj;
    pTarget.trans := [19,21.0,0];
    MoveL pTarget,vSpeed,z0,tTool\WObj:=wWobj;
    pTarget.trans := [18,16.0,0];
    MoveL pTarget,vSpeed,z0,tTool\WObj:=wWobj;
    pTarget.trans := [17,14.0,0];
    MoveL pTarget,vSpeed,z0,tTool\WObj:=wWobj;
    pTarget.trans := [15,12.0,0];
    MoveL pTarget,vSpeed,z0,tTool\WObj:=wWobj;
    pTarget.trans := [12,11.0,0];
    MoveL pTarget,vSpeed,z0,tTool\WObj:=wWobj;
    pTarget.trans := [8,11.0,0];
    MoveL pTarget,vSpeed,z0,tTool\WObj:=wWobj;
    pTarget.trans := [5,12.0,0];
    MoveL pTarget,vSpeed,z0,tTool\WObj:=wWobj;
    pTarget.trans := [3,14.0,0];
    MoveL pTarget,vSpeed,z0,tTool\WObj:=wWobj;
    pTarget.trans := [2,16.0,0];
    MoveL pTarget,vSpeed,z0,tTool\WObj:=wWobj;
    pTarget.trans := [2,18.0,0];
    MoveL pTarget,vSpeed,fine,tTool\WObj:=wWobj;
    Reset do_pen;
    MoveL RelTool(pTarget,0,0,-2),vSpeed,z0,tTool\WObj:=wWobj;
    wWobj.oframe.trans.x := wWobj.oframe.trans.x + 19;
ENDPROC
  ! Character: H
  PROC char_upperH()
    VAR robtarget pTarget;
    pTarget := refTarget;
    pTarget.trans := [7,25.0,0];
    MoveL pTarget,vSpeed,fine,tTool\WObj:=wWobj;
    Set do_pen;
    pTarget.trans := [5,26.0,0];
    MoveL pTarget,vSpeed,z0,tTool\WObj:=wWobj;
    pTarget.trans := [4,28.0,0];
    MoveL pTarget,vSpeed,z0,tTool\WObj:=wWobj;
    pTarget.trans := [4,29.0,0];
    MoveL pTarget,vSpeed,z0,tTool\WObj:=wWobj;
    pTarget.trans := [5,31.0,0];
    MoveL pTarget,vSpeed,z0,tTool\WObj:=wWobj;
    pTarget.trans := [7,32.0,0];
    MoveL pTarget,vSpeed,z0,tTool\WObj:=wWobj;
    pTarget.trans := [8,32.0,0];
    MoveL pTarget,vSpeed,z0,tTool\WObj:=wWobj;
    pTarget.trans := [10,31.0,0];
    MoveL pTarget,vSpeed,z0,tTool\WObj:=wWobj;
    pTarget.trans := [11,29.0,0];
    MoveL pTarget,vSpeed,z0,tTool\WObj:=wWobj;
    pTarget.trans := [11,27.0,0];
    MoveL pTarget,vSpeed,z0,tTool\WObj:=wWobj;
    pTarget.trans := [10,23.0,0];
    MoveL pTarget,vSpeed,z0,tTool\WObj:=wWobj;
    pTarget.trans := [8,17.0,0];
    MoveL pTarget,vSpeed,z0,tTool\WObj:=wWobj;
    pTarget.trans := [6,13.0,0];
    MoveL pTarget,vSpeed,z0,tTool\WObj:=wWobj;
    pTarget.trans := [4,11.0,0];
    MoveL pTarget,vSpeed,z0,tTool\WObj:=wWobj;
    pTarget.trans := [2,11.0,0];
    MoveL pTarget,vSpeed,z0,tTool\WObj:=wWobj;
    pTarget.trans := [1,12.0,0];
    MoveL pTarget,vSpeed,z0,tTool\WObj:=wWobj;
    pTarget.trans := [1,14.0,0];
    MoveL pTarget,vSpeed,fine,tTool\WObj:=wWobj;
    Reset do_pen;
    MoveL RelTool(pTarget,0,0,-2),vSpeed,z0,tTool\WObj:=wWobj;
    pTarget.trans := [7,20.0,0];
    MoveL pTarget,vSpeed,fine,tTool\WObj:=wWobj;
    Set do_pen;
    pTarget.trans := [16,23.0,0];
    MoveL pTarget,vSpeed,z0,tTool\WObj:=wWobj;
    pTarget.trans := [18,24.0,0];
    MoveL pTarget,vSpeed,z0,tTool\WObj:=wWobj;
    pTarget.trans := [21,26.0,0];
    MoveL pTarget,vSpeed,z0,tTool\WObj:=wWobj;
    pTarget.trans := [23,28.0,0];
    MoveL pTarget,vSpeed,z0,tTool\WObj:=wWobj;
    pTarget.trans := [24,30.0,0];
    MoveL pTarget,vSpeed,z0,tTool\WObj:=wWobj;
    pTarget.trans := [24,31.0,0];
    MoveL pTarget,vSpeed,z0,tTool\WObj:=wWobj;
    pTarget.trans := [23,32.0,0];
    MoveL pTarget,vSpeed,z0,tTool\WObj:=wWobj;
    pTarget.trans := [22,32.0,0];
    MoveL pTarget,vSpeed,z0,tTool\WObj:=wWobj;
    pTarget.trans := [20,30.0,0];
    MoveL pTarget,vSpeed,z0,tTool\WObj:=wWobj;
    pTarget.trans := [18,26.0,0];
    MoveL pTarget,vSpeed,z0,tTool\WObj:=wWobj;
    pTarget.trans := [16,20.0,0];
    MoveL pTarget,vSpeed,z0,tTool\WObj:=wWobj;
    pTarget.trans := [15,15.0,0];
    MoveL pTarget,vSpeed,z0,tTool\WObj:=wWobj;
    pTarget.trans := [15,12.0,0];
    MoveL pTarget,vSpeed,z0,tTool\WObj:=wWobj;
    pTarget.trans := [16,11.0,0];
    MoveL pTarget,vSpeed,z0,tTool\WObj:=wWobj;
    pTarget.trans := [17,11.0,0];
    MoveL pTarget,vSpeed,z0,tTool\WObj:=wWobj;
    pTarget.trans := [19,12.0,0];
    MoveL pTarget,vSpeed,z0,tTool\WObj:=wWobj;
    pTarget.trans := [20,13.0,0];
    MoveL pTarget,vSpeed,z0,tTool\WObj:=wWobj;
    pTarget.trans := [22,16.0,0];
    MoveL pTarget,vSpeed,fine,tTool\WObj:=wWobj;
    Reset do_pen;
    MoveL RelTool(pTarget,0,0,-2),vSpeed,z0,tTool\WObj:=wWobj;
    wWobj.oframe.trans.x := wWobj.oframe.trans.x + 23;
ENDPROC
  ! Character: I
  PROC char_upperI()
    VAR robtarget pTarget;
    pTarget := refTarget;
    pTarget.trans := [14,16.0,0];
    MoveL pTarget,vSpeed,fine,tTool\WObj:=wWobj;
    Set do_pen;
    pTarget.trans := [12,18.0,0];
    MoveL pTarget,vSpeed,z0,tTool\WObj:=wWobj;
    pTarget.trans := [10,21.0,0];
    MoveL pTarget,vSpeed,z0,tTool\WObj:=wWobj;
    pTarget.trans := [9,23.0,0];
    MoveL pTarget,vSpeed,z0,tTool\WObj:=wWobj;
    pTarget.trans := [8,26.0,0];
    MoveL pTarget,vSpeed,z0,tTool\WObj:=wWobj;
    pTarget.trans := [8,29.0,0];
    MoveL pTarget,vSpeed,z0,tTool\WObj:=wWobj;
    pTarget.trans := [9,31.0,0];
    MoveL pTarget,vSpeed,z0,tTool\WObj:=wWobj;
    pTarget.trans := [10,32.0,0];
    MoveL pTarget,vSpeed,z0,tTool\WObj:=wWobj;
    pTarget.trans := [12,32.0,0];
    MoveL pTarget,vSpeed,z0,tTool\WObj:=wWobj;
    pTarget.trans := [13,31.0,0];
    MoveL pTarget,vSpeed,z0,tTool\WObj:=wWobj;
    pTarget.trans := [14,29.0,0];
    MoveL pTarget,vSpeed,z0,tTool\WObj:=wWobj;
    pTarget.trans := [14,26.0,0];
    MoveL pTarget,vSpeed,z0,tTool\WObj:=wWobj;
    pTarget.trans := [13,21.0,0];
    MoveL pTarget,vSpeed,z0,tTool\WObj:=wWobj;
    pTarget.trans := [11,16.0,0];
    MoveL pTarget,vSpeed,z0,tTool\WObj:=wWobj;
    pTarget.trans := [10,14.0,0];
    MoveL pTarget,vSpeed,z0,tTool\WObj:=wWobj;
    pTarget.trans := [8,12.0,0];
    MoveL pTarget,vSpeed,z0,tTool\WObj:=wWobj;
    pTarget.trans := [6,11.0,0];
    MoveL pTarget,vSpeed,z0,tTool\WObj:=wWobj;
    pTarget.trans := [4,11.0,0];
    MoveL pTarget,vSpeed,z0,tTool\WObj:=wWobj;
    pTarget.trans := [2,12.0,0];
    MoveL pTarget,vSpeed,z0,tTool\WObj:=wWobj;
    pTarget.trans := [1,14.0,0];
    MoveL pTarget,vSpeed,z0,tTool\WObj:=wWobj;
    pTarget.trans := [1,16.0,0];
    MoveL pTarget,vSpeed,z0,tTool\WObj:=wWobj;
    pTarget.trans := [2,17.0,0];
    MoveL pTarget,vSpeed,z0,tTool\WObj:=wWobj;
    pTarget.trans := [4,17.0,0];
    MoveL pTarget,vSpeed,z0,tTool\WObj:=wWobj;
    pTarget.trans := [6,16.0,0];
    MoveL pTarget,vSpeed,fine,tTool\WObj:=wWobj;
    Reset do_pen;
    MoveL RelTool(pTarget,0,0,-2),vSpeed,z0,tTool\WObj:=wWobj;
    wWobj.oframe.trans.x := wWobj.oframe.trans.x + 13;
ENDPROC
  ! Character: J
  PROC char_upperJ()
    VAR robtarget pTarget;
    pTarget := refTarget;
    pTarget.trans := [10,8.0,0];
    MoveL pTarget,vSpeed,fine,tTool\WObj:=wWobj;
    Set do_pen;
    pTarget.trans := [8,11.0,0];
    MoveL pTarget,vSpeed,z0,tTool\WObj:=wWobj;
    pTarget.trans := [6,16.0,0];
    MoveL pTarget,vSpeed,z0,tTool\WObj:=wWobj;
    pTarget.trans := [5,22.0,0];
    MoveL pTarget,vSpeed,z0,tTool\WObj:=wWobj;
    pTarget.trans := [5,28.0,0];
    MoveL pTarget,vSpeed,z0,tTool\WObj:=wWobj;
    pTarget.trans := [6,31.0,0];
    MoveL pTarget,vSpeed,z0,tTool\WObj:=wWobj;
    pTarget.trans := [8,32.0,0];
    MoveL pTarget,vSpeed,z0,tTool\WObj:=wWobj;
    pTarget.trans := [10,32.0,0];
    MoveL pTarget,vSpeed,z0,tTool\WObj:=wWobj;
    pTarget.trans := [11,31.0,0];
    MoveL pTarget,vSpeed,z0,tTool\WObj:=wWobj;
    pTarget.trans := [12,28.0,0];
    MoveL pTarget,vSpeed,z0,tTool\WObj:=wWobj;
    pTarget.trans := [12,25.0,0];
    MoveL pTarget,vSpeed,z0,tTool\WObj:=wWobj;
    pTarget.trans := [11,20.0,0];
    MoveL pTarget,vSpeed,z0,tTool\WObj:=wWobj;
    pTarget.trans := [8,11.0,0];
    MoveL pTarget,vSpeed,z0,tTool\WObj:=wWobj;
    pTarget.trans := [6,5.0,0];
    MoveL pTarget,vSpeed,z0,tTool\WObj:=wWobj;
    pTarget.trans := [5,2.0,0];
    MoveL pTarget,vSpeed,z0,tTool\WObj:=wWobj;
    pTarget.trans := [4,0.0,0];
    MoveL pTarget,vSpeed,z0,tTool\WObj:=wWobj;
    pTarget.trans := [2,-1.0,0];
    MoveL pTarget,vSpeed,z0,tTool\WObj:=wWobj;
    pTarget.trans := [1,0.0,0];
    MoveL pTarget,vSpeed,z0,tTool\WObj:=wWobj;
    pTarget.trans := [1,2.0,0];
    MoveL pTarget,vSpeed,z0,tTool\WObj:=wWobj;
    pTarget.trans := [2,5.0,0];
    MoveL pTarget,vSpeed,z0,tTool\WObj:=wWobj;
    pTarget.trans := [4,8.0,0];
    MoveL pTarget,vSpeed,z0,tTool\WObj:=wWobj;
    pTarget.trans := [6,10.0,0];
    MoveL pTarget,vSpeed,z0,tTool\WObj:=wWobj;
    pTarget.trans := [9,12.0,0];
    MoveL pTarget,vSpeed,z0,tTool\WObj:=wWobj;
    pTarget.trans := [13,14.0,0];
    MoveL pTarget,vSpeed,fine,tTool\WObj:=wWobj;
    Reset do_pen;
    MoveL RelTool(pTarget,0,0,-2),vSpeed,z0,tTool\WObj:=wWobj;
    wWobj.oframe.trans.x := wWobj.oframe.trans.x + 12;
ENDPROC
  ! Character: K
  PROC char_upperK()
    VAR robtarget pTarget;
    pTarget := refTarget;
    pTarget.trans := [7,25.0,0];
    MoveL pTarget,vSpeed,fine,tTool\WObj:=wWobj;
    Set do_pen;
    pTarget.trans := [5,26.0,0];
    MoveL pTarget,vSpeed,z0,tTool\WObj:=wWobj;
    pTarget.trans := [4,28.0,0];
    MoveL pTarget,vSpeed,z0,tTool\WObj:=wWobj;
    pTarget.trans := [4,29.0,0];
    MoveL pTarget,vSpeed,z0,tTool\WObj:=wWobj;
    pTarget.trans := [5,31.0,0];
    MoveL pTarget,vSpeed,z0,tTool\WObj:=wWobj;
    pTarget.trans := [7,32.0,0];
    MoveL pTarget,vSpeed,z0,tTool\WObj:=wWobj;
    pTarget.trans := [8,32.0,0];
    MoveL pTarget,vSpeed,z0,tTool\WObj:=wWobj;
    pTarget.trans := [10,31.0,0];
    MoveL pTarget,vSpeed,z0,tTool\WObj:=wWobj;
    pTarget.trans := [11,29.0,0];
    MoveL pTarget,vSpeed,z0,tTool\WObj:=wWobj;
    pTarget.trans := [11,27.0,0];
    MoveL pTarget,vSpeed,z0,tTool\WObj:=wWobj;
    pTarget.trans := [10,23.0,0];
    MoveL pTarget,vSpeed,z0,tTool\WObj:=wWobj;
    pTarget.trans := [8,17.0,0];
    MoveL pTarget,vSpeed,z0,tTool\WObj:=wWobj;
    pTarget.trans := [6,13.0,0];
    MoveL pTarget,vSpeed,z0,tTool\WObj:=wWobj;
    pTarget.trans := [4,11.0,0];
    MoveL pTarget,vSpeed,z0,tTool\WObj:=wWobj;
    pTarget.trans := [2,11.0,0];
    MoveL pTarget,vSpeed,z0,tTool\WObj:=wWobj;
    pTarget.trans := [1,12.0,0];
    MoveL pTarget,vSpeed,z0,tTool\WObj:=wWobj;
    pTarget.trans := [1,14.0,0];
    MoveL pTarget,vSpeed,fine,tTool\WObj:=wWobj;
    Reset do_pen;
    MoveL RelTool(pTarget,0,0,-2),vSpeed,z0,tTool\WObj:=wWobj;
    pTarget.trans := [24,29.0,0];
    MoveL pTarget,vSpeed,fine,tTool\WObj:=wWobj;
    Set do_pen;
    pTarget.trans := [24,31.0,0];
    MoveL pTarget,vSpeed,z0,tTool\WObj:=wWobj;
    pTarget.trans := [23,32.0,0];
    MoveL pTarget,vSpeed,z0,tTool\WObj:=wWobj;
    pTarget.trans := [22,32.0,0];
    MoveL pTarget,vSpeed,z0,tTool\WObj:=wWobj;
    pTarget.trans := [20,31.0,0];
    MoveL pTarget,vSpeed,z0,tTool\WObj:=wWobj;
    pTarget.trans := [18,29.0,0];
    MoveL pTarget,vSpeed,z0,tTool\WObj:=wWobj;
    pTarget.trans := [16,26.0,0];
    MoveL pTarget,vSpeed,z0,tTool\WObj:=wWobj;
    pTarget.trans := [14,24.0,0];
    MoveL pTarget,vSpeed,z0,tTool\WObj:=wWobj;
    pTarget.trans := [12,23.0,0];
    MoveL pTarget,vSpeed,z0,tTool\WObj:=wWobj;
    pTarget.trans := [10,23.0,0];
    MoveL pTarget,vSpeed,fine,tTool\WObj:=wWobj;
    Reset do_pen;
    MoveL RelTool(pTarget,0,0,-2),vSpeed,z0,tTool\WObj:=wWobj;
    pTarget.trans := [12,23.0,0];
    MoveL pTarget,vSpeed,fine,tTool\WObj:=wWobj;
    Set do_pen;
    pTarget.trans := [13,21.0,0];
    MoveL pTarget,vSpeed,z0,tTool\WObj:=wWobj;
    pTarget.trans := [13,14.0,0];
    MoveL pTarget,vSpeed,z0,tTool\WObj:=wWobj;
    pTarget.trans := [14,12.0,0];
    MoveL pTarget,vSpeed,z0,tTool\WObj:=wWobj;
    pTarget.trans := [15,11.0,0];
    MoveL pTarget,vSpeed,z0,tTool\WObj:=wWobj;
    pTarget.trans := [16,11.0,0];
    MoveL pTarget,vSpeed,z0,tTool\WObj:=wWobj;
    pTarget.trans := [18,12.0,0];
    MoveL pTarget,vSpeed,z0,tTool\WObj:=wWobj;
    pTarget.trans := [19,13.0,0];
    MoveL pTarget,vSpeed,z0,tTool\WObj:=wWobj;
    pTarget.trans := [21,16.0,0];
    MoveL pTarget,vSpeed,fine,tTool\WObj:=wWobj;
    Reset do_pen;
    MoveL RelTool(pTarget,0,0,-2),vSpeed,z0,tTool\WObj:=wWobj;
    wWobj.oframe.trans.x := wWobj.oframe.trans.x + 23;
ENDPROC
  ! Character: L
  PROC char_upperL()
    VAR robtarget pTarget;
    pTarget := refTarget;
    pTarget.trans := [4,20.0,0];
    MoveL pTarget,vSpeed,fine,tTool\WObj:=wWobj;
    Set do_pen;
    pTarget.trans := [6,20.0,0];
    MoveL pTarget,vSpeed,z0,tTool\WObj:=wWobj;
    pTarget.trans := [10,21.0,0];
    MoveL pTarget,vSpeed,z0,tTool\WObj:=wWobj;
    pTarget.trans := [13,23.0,0];
    MoveL pTarget,vSpeed,z0,tTool\WObj:=wWobj;
    pTarget.trans := [15,25.0,0];
    MoveL pTarget,vSpeed,z0,tTool\WObj:=wWobj;
    pTarget.trans := [16,27.0,0];
    MoveL pTarget,vSpeed,z0,tTool\WObj:=wWobj;
    pTarget.trans := [16,30.0,0];
    MoveL pTarget,vSpeed,z0,tTool\WObj:=wWobj;
    pTarget.trans := [15,32.0,0];
    MoveL pTarget,vSpeed,z0,tTool\WObj:=wWobj;
    pTarget.trans := [13,32.0,0];
    MoveL pTarget,vSpeed,z0,tTool\WObj:=wWobj;
    pTarget.trans := [12,31.0,0];
    MoveL pTarget,vSpeed,z0,tTool\WObj:=wWobj;
    pTarget.trans := [11,29.0,0];
    MoveL pTarget,vSpeed,z0,tTool\WObj:=wWobj;
    pTarget.trans := [10,24.0,0];
    MoveL pTarget,vSpeed,z0,tTool\WObj:=wWobj;
    pTarget.trans := [9,19.0,0];
    MoveL pTarget,vSpeed,z0,tTool\WObj:=wWobj;
    pTarget.trans := [8,16.0,0];
    MoveL pTarget,vSpeed,z0,tTool\WObj:=wWobj;
    pTarget.trans := [7,14.0,0];
    MoveL pTarget,vSpeed,z0,tTool\WObj:=wWobj;
    pTarget.trans := [5,12.0,0];
    MoveL pTarget,vSpeed,z0,tTool\WObj:=wWobj;
    pTarget.trans := [3,11.0,0];
    MoveL pTarget,vSpeed,z0,tTool\WObj:=wWobj;
    pTarget.trans := [1,11.0,0];
    MoveL pTarget,vSpeed,z0,tTool\WObj:=wWobj;
    pTarget.trans := [0,12.0,0];
    MoveL pTarget,vSpeed,z0,tTool\WObj:=wWobj;
    pTarget.trans := [0,14.0,0];
    MoveL pTarget,vSpeed,z0,tTool\WObj:=wWobj;
    pTarget.trans := [1,15.0,0];
    MoveL pTarget,vSpeed,z0,tTool\WObj:=wWobj;
    pTarget.trans := [3,15.0,0];
    MoveL pTarget,vSpeed,z0,tTool\WObj:=wWobj;
    pTarget.trans := [5,14.0,0];
    MoveL pTarget,vSpeed,z0,tTool\WObj:=wWobj;
    pTarget.trans := [8,12.0,0];
    MoveL pTarget,vSpeed,z0,tTool\WObj:=wWobj;
    pTarget.trans := [11,11.0,0];
    MoveL pTarget,vSpeed,z0,tTool\WObj:=wWobj;
    pTarget.trans := [13,11.0,0];
    MoveL pTarget,vSpeed,z0,tTool\WObj:=wWobj;
    pTarget.trans := [16,12.0,0];
    MoveL pTarget,vSpeed,z0,tTool\WObj:=wWobj;
    pTarget.trans := [18,14.0,0];
    MoveL pTarget,vSpeed,fine,tTool\WObj:=wWobj;
    Reset do_pen;
    MoveL RelTool(pTarget,0,0,-2),vSpeed,z0,tTool\WObj:=wWobj;
    wWobj.oframe.trans.x := wWobj.oframe.trans.x + 18;
ENDPROC
  ! Character: M
  PROC char_upperM()
    VAR robtarget pTarget;
    pTarget := refTarget;
    pTarget.trans := [5,25.0,0];
    MoveL pTarget,vSpeed,fine,tTool\WObj:=wWobj;
    Set do_pen;
    pTarget.trans := [3,26.0,0];
    MoveL pTarget,vSpeed,z0,tTool\WObj:=wWobj;
    pTarget.trans := [2,28.0,0];
    MoveL pTarget,vSpeed,z0,tTool\WObj:=wWobj;
    pTarget.trans := [2,29.0,0];
    MoveL pTarget,vSpeed,z0,tTool\WObj:=wWobj;
    pTarget.trans := [3,31.0,0];
    MoveL pTarget,vSpeed,z0,tTool\WObj:=wWobj;
    pTarget.trans := [5,32.0,0];
    MoveL pTarget,vSpeed,z0,tTool\WObj:=wWobj;
    pTarget.trans := [6,32.0,0];
    MoveL pTarget,vSpeed,z0,tTool\WObj:=wWobj;
    pTarget.trans := [8,31.0,0];
    MoveL pTarget,vSpeed,z0,tTool\WObj:=wWobj;
    pTarget.trans := [9,29.0,0];
    MoveL pTarget,vSpeed,z0,tTool\WObj:=wWobj;
    pTarget.trans := [9,27.0,0];
    MoveL pTarget,vSpeed,z0,tTool\WObj:=wWobj;
    pTarget.trans := [8,22.0,0];
    MoveL pTarget,vSpeed,z0,tTool\WObj:=wWobj;
    pTarget.trans := [7,18.0,0];
    MoveL pTarget,vSpeed,z0,tTool\WObj:=wWobj;
    pTarget.trans := [5,11.0,0];
    MoveL pTarget,vSpeed,fine,tTool\WObj:=wWobj;
    Reset do_pen;
    MoveL RelTool(pTarget,0,0,-2),vSpeed,z0,tTool\WObj:=wWobj;
    pTarget.trans := [7,18.0,0];
    MoveL pTarget,vSpeed,fine,tTool\WObj:=wWobj;
    Set do_pen;
    pTarget.trans := [10,26.0,0];
    MoveL pTarget,vSpeed,z0,tTool\WObj:=wWobj;
    pTarget.trans := [12,30.0,0];
    MoveL pTarget,vSpeed,z0,tTool\WObj:=wWobj;
    pTarget.trans := [13,31.0,0];
    MoveL pTarget,vSpeed,z0,tTool\WObj:=wWobj;
    pTarget.trans := [15,32.0,0];
    MoveL pTarget,vSpeed,z0,tTool\WObj:=wWobj;
    pTarget.trans := [16,32.0,0];
    MoveL pTarget,vSpeed,z0,tTool\WObj:=wWobj;
    pTarget.trans := [18,31.0,0];
    MoveL pTarget,vSpeed,z0,tTool\WObj:=wWobj;
    pTarget.trans := [19,29.0,0];
    MoveL pTarget,vSpeed,z0,tTool\WObj:=wWobj;
    pTarget.trans := [19,27.0,0];
    MoveL pTarget,vSpeed,z0,tTool\WObj:=wWobj;
    pTarget.trans := [18,22.0,0];
    MoveL pTarget,vSpeed,z0,tTool\WObj:=wWobj;
    pTarget.trans := [17,18.0,0];
    MoveL pTarget,vSpeed,z0,tTool\WObj:=wWobj;
    pTarget.trans := [15,11.0,0];
    MoveL pTarget,vSpeed,fine,tTool\WObj:=wWobj;
    Reset do_pen;
    MoveL RelTool(pTarget,0,0,-2),vSpeed,z0,tTool\WObj:=wWobj;
    pTarget.trans := [17,18.0,0];
    MoveL pTarget,vSpeed,fine,tTool\WObj:=wWobj;
    Set do_pen;
    pTarget.trans := [20,26.0,0];
    MoveL pTarget,vSpeed,z0,tTool\WObj:=wWobj;
    pTarget.trans := [22,30.0,0];
    MoveL pTarget,vSpeed,z0,tTool\WObj:=wWobj;
    pTarget.trans := [23,31.0,0];
    MoveL pTarget,vSpeed,z0,tTool\WObj:=wWobj;
    pTarget.trans := [25,32.0,0];
    MoveL pTarget,vSpeed,z0,tTool\WObj:=wWobj;
    pTarget.trans := [26,32.0,0];
    MoveL pTarget,vSpeed,z0,tTool\WObj:=wWobj;
    pTarget.trans := [28,31.0,0];
    MoveL pTarget,vSpeed,z0,tTool\WObj:=wWobj;
    pTarget.trans := [29,29.0,0];
    MoveL pTarget,vSpeed,z0,tTool\WObj:=wWobj;
    pTarget.trans := [29,27.0,0];
    MoveL pTarget,vSpeed,z0,tTool\WObj:=wWobj;
    pTarget.trans := [28,22.0,0];
    MoveL pTarget,vSpeed,z0,tTool\WObj:=wWobj;
    pTarget.trans := [26,15.0,0];
    MoveL pTarget,vSpeed,z0,tTool\WObj:=wWobj;
    pTarget.trans := [26,12.0,0];
    MoveL pTarget,vSpeed,z0,tTool\WObj:=wWobj;
    pTarget.trans := [27,11.0,0];
    MoveL pTarget,vSpeed,z0,tTool\WObj:=wWobj;
    pTarget.trans := [28,11.0,0];
    MoveL pTarget,vSpeed,z0,tTool\WObj:=wWobj;
    pTarget.trans := [30,12.0,0];
    MoveL pTarget,vSpeed,z0,tTool\WObj:=wWobj;
    pTarget.trans := [31,13.0,0];
    MoveL pTarget,vSpeed,z0,tTool\WObj:=wWobj;
    pTarget.trans := [33,16.0,0];
    MoveL pTarget,vSpeed,fine,tTool\WObj:=wWobj;
    Reset do_pen;
    MoveL RelTool(pTarget,0,0,-2),vSpeed,z0,tTool\WObj:=wWobj;
    wWobj.oframe.trans.x := wWobj.oframe.trans.x + 31;
ENDPROC
  ! Character: N
  PROC char_upperN()
    VAR robtarget pTarget;
    pTarget := refTarget;
    pTarget.trans := [5,25.0,0];
    MoveL pTarget,vSpeed,fine,tTool\WObj:=wWobj;
    Set do_pen;
    pTarget.trans := [3,26.0,0];
    MoveL pTarget,vSpeed,z0,tTool\WObj:=wWobj;
    pTarget.trans := [2,28.0,0];
    MoveL pTarget,vSpeed,z0,tTool\WObj:=wWobj;
    pTarget.trans := [2,29.0,0];
    MoveL pTarget,vSpeed,z0,tTool\WObj:=wWobj;
    pTarget.trans := [3,31.0,0];
    MoveL pTarget,vSpeed,z0,tTool\WObj:=wWobj;
    pTarget.trans := [5,32.0,0];
    MoveL pTarget,vSpeed,z0,tTool\WObj:=wWobj;
    pTarget.trans := [6,32.0,0];
    MoveL pTarget,vSpeed,z0,tTool\WObj:=wWobj;
    pTarget.trans := [8,31.0,0];
    MoveL pTarget,vSpeed,z0,tTool\WObj:=wWobj;
    pTarget.trans := [9,29.0,0];
    MoveL pTarget,vSpeed,z0,tTool\WObj:=wWobj;
    pTarget.trans := [9,27.0,0];
    MoveL pTarget,vSpeed,z0,tTool\WObj:=wWobj;
    pTarget.trans := [8,22.0,0];
    MoveL pTarget,vSpeed,z0,tTool\WObj:=wWobj;
    pTarget.trans := [7,18.0,0];
    MoveL pTarget,vSpeed,z0,tTool\WObj:=wWobj;
    pTarget.trans := [5,11.0,0];
    MoveL pTarget,vSpeed,fine,tTool\WObj:=wWobj;
    Reset do_pen;
    MoveL RelTool(pTarget,0,0,-2),vSpeed,z0,tTool\WObj:=wWobj;
    pTarget.trans := [7,18.0,0];
    MoveL pTarget,vSpeed,fine,tTool\WObj:=wWobj;
    Set do_pen;
    pTarget.trans := [10,26.0,0];
    MoveL pTarget,vSpeed,z0,tTool\WObj:=wWobj;
    pTarget.trans := [12,30.0,0];
    MoveL pTarget,vSpeed,z0,tTool\WObj:=wWobj;
    pTarget.trans := [13,31.0,0];
    MoveL pTarget,vSpeed,z0,tTool\WObj:=wWobj;
    pTarget.trans := [15,32.0,0];
    MoveL pTarget,vSpeed,z0,tTool\WObj:=wWobj;
    pTarget.trans := [17,32.0,0];
    MoveL pTarget,vSpeed,z0,tTool\WObj:=wWobj;
    pTarget.trans := [19,31.0,0];
    MoveL pTarget,vSpeed,z0,tTool\WObj:=wWobj;
    pTarget.trans := [20,29.0,0];
    MoveL pTarget,vSpeed,z0,tTool\WObj:=wWobj;
    pTarget.trans := [20,27.0,0];
    MoveL pTarget,vSpeed,z0,tTool\WObj:=wWobj;
    pTarget.trans := [19,22.0,0];
    MoveL pTarget,vSpeed,z0,tTool\WObj:=wWobj;
    pTarget.trans := [17,15.0,0];
    MoveL pTarget,vSpeed,z0,tTool\WObj:=wWobj;
    pTarget.trans := [17,12.0,0];
    MoveL pTarget,vSpeed,z0,tTool\WObj:=wWobj;
    pTarget.trans := [18,11.0,0];
    MoveL pTarget,vSpeed,z0,tTool\WObj:=wWobj;
    pTarget.trans := [19,11.0,0];
    MoveL pTarget,vSpeed,z0,tTool\WObj:=wWobj;
    pTarget.trans := [21,12.0,0];
    MoveL pTarget,vSpeed,z0,tTool\WObj:=wWobj;
    pTarget.trans := [22,13.0,0];
    MoveL pTarget,vSpeed,z0,tTool\WObj:=wWobj;
    pTarget.trans := [24,16.0,0];
    MoveL pTarget,vSpeed,fine,tTool\WObj:=wWobj;
    Reset do_pen;
    MoveL RelTool(pTarget,0,0,-2),vSpeed,z0,tTool\WObj:=wWobj;
    wWobj.oframe.trans.x := wWobj.oframe.trans.x + 22;
ENDPROC
  ! Character: O
  PROC char_upperO()
    VAR robtarget pTarget;
    pTarget := refTarget;
    pTarget.trans := [12,32.0,0];
    MoveL pTarget,vSpeed,fine,tTool\WObj:=wWobj;
    Set do_pen;
    pTarget.trans := [9,31.0,0];
    MoveL pTarget,vSpeed,z0,tTool\WObj:=wWobj;
    pTarget.trans := [7,29.0,0];
    MoveL pTarget,vSpeed,z0,tTool\WObj:=wWobj;
    pTarget.trans := [5,26.0,0];
    MoveL pTarget,vSpeed,z0,tTool\WObj:=wWobj;
    pTarget.trans := [4,24.0,0];
    MoveL pTarget,vSpeed,z0,tTool\WObj:=wWobj;
    pTarget.trans := [3,20.0,0];
    MoveL pTarget,vSpeed,z0,tTool\WObj:=wWobj;
    pTarget.trans := [3,16.0,0];
    MoveL pTarget,vSpeed,z0,tTool\WObj:=wWobj;
    pTarget.trans := [4,13.0,0];
    MoveL pTarget,vSpeed,z0,tTool\WObj:=wWobj;
    pTarget.trans := [5,12.0,0];
    MoveL pTarget,vSpeed,z0,tTool\WObj:=wWobj;
    pTarget.trans := [7,11.0,0];
    MoveL pTarget,vSpeed,z0,tTool\WObj:=wWobj;
    pTarget.trans := [9,11.0,0];
    MoveL pTarget,vSpeed,z0,tTool\WObj:=wWobj;
    pTarget.trans := [12,12.0,0];
    MoveL pTarget,vSpeed,z0,tTool\WObj:=wWobj;
    pTarget.trans := [14,14.0,0];
    MoveL pTarget,vSpeed,z0,tTool\WObj:=wWobj;
    pTarget.trans := [16,17.0,0];
    MoveL pTarget,vSpeed,z0,tTool\WObj:=wWobj;
    pTarget.trans := [17,19.0,0];
    MoveL pTarget,vSpeed,z0,tTool\WObj:=wWobj;
    pTarget.trans := [18,23.0,0];
    MoveL pTarget,vSpeed,z0,tTool\WObj:=wWobj;
    pTarget.trans := [18,27.0,0];
    MoveL pTarget,vSpeed,z0,tTool\WObj:=wWobj;
    pTarget.trans := [17,30.0,0];
    MoveL pTarget,vSpeed,z0,tTool\WObj:=wWobj;
    pTarget.trans := [16,31.0,0];
    MoveL pTarget,vSpeed,z0,tTool\WObj:=wWobj;
    pTarget.trans := [14,32.0,0];
    MoveL pTarget,vSpeed,z0,tTool\WObj:=wWobj;
    pTarget.trans := [12,32.0,0];
    MoveL pTarget,vSpeed,z0,tTool\WObj:=wWobj;
    pTarget.trans := [10,30.0,0];
    MoveL pTarget,vSpeed,z0,tTool\WObj:=wWobj;
    pTarget.trans := [10,27.0,0];
    MoveL pTarget,vSpeed,z0,tTool\WObj:=wWobj;
    pTarget.trans := [11,24.0,0];
    MoveL pTarget,vSpeed,z0,tTool\WObj:=wWobj;
    pTarget.trans := [13,21.0,0];
    MoveL pTarget,vSpeed,z0,tTool\WObj:=wWobj;
    pTarget.trans := [15,19.0,0];
    MoveL pTarget,vSpeed,z0,tTool\WObj:=wWobj;
    pTarget.trans := [18,17.0,0];
    MoveL pTarget,vSpeed,z0,tTool\WObj:=wWobj;
    pTarget.trans := [20,16.0,0];
    MoveL pTarget,vSpeed,fine,tTool\WObj:=wWobj;
    Reset do_pen;
    MoveL RelTool(pTarget,0,0,-2),vSpeed,z0,tTool\WObj:=wWobj;
    wWobj.oframe.trans.x := wWobj.oframe.trans.x + 17;
ENDPROC
  ! Character: P
  PROC char_upperP()
    VAR robtarget pTarget;
    pTarget := refTarget;
    pTarget.trans := [13,30.0,0];
    MoveL pTarget,vSpeed,fine,tTool\WObj:=wWobj;
    Set do_pen;
    pTarget.trans := [14,29.0,0];
    MoveL pTarget,vSpeed,z0,tTool\WObj:=wWobj;
    pTarget.trans := [14,26.0,0];
    MoveL pTarget,vSpeed,z0,tTool\WObj:=wWobj;
    pTarget.trans := [13,22.0,0];
    MoveL pTarget,vSpeed,z0,tTool\WObj:=wWobj;
    pTarget.trans := [12,19.0,0];
    MoveL pTarget,vSpeed,z0,tTool\WObj:=wWobj;
    pTarget.trans := [11,17.0,0];
    MoveL pTarget,vSpeed,z0,tTool\WObj:=wWobj;
    pTarget.trans := [9,14.0,0];
    MoveL pTarget,vSpeed,z0,tTool\WObj:=wWobj;
    pTarget.trans := [7,12.0,0];
    MoveL pTarget,vSpeed,z0,tTool\WObj:=wWobj;
    pTarget.trans := [5,11.0,0];
    MoveL pTarget,vSpeed,z0,tTool\WObj:=wWobj;
    pTarget.trans := [4,11.0,0];
    MoveL pTarget,vSpeed,z0,tTool\WObj:=wWobj;
    pTarget.trans := [3,12.0,0];
    MoveL pTarget,vSpeed,z0,tTool\WObj:=wWobj;
    pTarget.trans := [3,15.0,0];
    MoveL pTarget,vSpeed,z0,tTool\WObj:=wWobj;
    pTarget.trans := [4,20.0,0];
    MoveL pTarget,vSpeed,z0,tTool\WObj:=wWobj;
    pTarget.trans := [5,23.0,0];
    MoveL pTarget,vSpeed,z0,tTool\WObj:=wWobj;
    pTarget.trans := [6,25.0,0];
    MoveL pTarget,vSpeed,z0,tTool\WObj:=wWobj;
    pTarget.trans := [8,28.0,0];
    MoveL pTarget,vSpeed,z0,tTool\WObj:=wWobj;
    pTarget.trans := [10,30.0,0];
    MoveL pTarget,vSpeed,z0,tTool\WObj:=wWobj;
    pTarget.trans := [12,31.0,0];
    MoveL pTarget,vSpeed,z0,tTool\WObj:=wWobj;
    pTarget.trans := [15,32.0,0];
    MoveL pTarget,vSpeed,z0,tTool\WObj:=wWobj;
    pTarget.trans := [20,32.0,0];
    MoveL pTarget,vSpeed,z0,tTool\WObj:=wWobj;
    pTarget.trans := [22,31.0,0];
    MoveL pTarget,vSpeed,z0,tTool\WObj:=wWobj;
    pTarget.trans := [23,30.0,0];
    MoveL pTarget,vSpeed,z0,tTool\WObj:=wWobj;
    pTarget.trans := [24,28.0,0];
    MoveL pTarget,vSpeed,z0,tTool\WObj:=wWobj;
    pTarget.trans := [24,25.0,0];
    MoveL pTarget,vSpeed,z0,tTool\WObj:=wWobj;
    pTarget.trans := [23,23.0,0];
    MoveL pTarget,vSpeed,z0,tTool\WObj:=wWobj;
    pTarget.trans := [22,22.0,0];
    MoveL pTarget,vSpeed,z0,tTool\WObj:=wWobj;
    pTarget.trans := [20,21.0,0];
    MoveL pTarget,vSpeed,z0,tTool\WObj:=wWobj;
    pTarget.trans := [17,21.0,0];
    MoveL pTarget,vSpeed,z0,tTool\WObj:=wWobj;
    pTarget.trans := [15,22.0,0];
    MoveL pTarget,vSpeed,z0,tTool\WObj:=wWobj;
    pTarget.trans := [14,23.0,0];
    MoveL pTarget,vSpeed,fine,tTool\WObj:=wWobj;
    Reset do_pen;
    MoveL RelTool(pTarget,0,0,-2),vSpeed,z0,tTool\WObj:=wWobj;
    wWobj.oframe.trans.x := wWobj.oframe.trans.x + 21;
ENDPROC
  ! Character: Q
  PROC char_upperQ()
    VAR robtarget pTarget;
    pTarget := refTarget;
    pTarget.trans := [13,26.0,0];
    MoveL pTarget,vSpeed,fine,tTool\WObj:=wWobj;
    Set do_pen;
    pTarget.trans := [12,24.0,0];
    MoveL pTarget,vSpeed,z0,tTool\WObj:=wWobj;
    pTarget.trans := [11,23.0,0];
    MoveL pTarget,vSpeed,z0,tTool\WObj:=wWobj;
    pTarget.trans := [9,22.0,0];
    MoveL pTarget,vSpeed,z0,tTool\WObj:=wWobj;
    pTarget.trans := [7,22.0,0];
    MoveL pTarget,vSpeed,z0,tTool\WObj:=wWobj;
    pTarget.trans := [6,24.0,0];
    MoveL pTarget,vSpeed,z0,tTool\WObj:=wWobj;
    pTarget.trans := [6,26.0,0];
    MoveL pTarget,vSpeed,z0,tTool\WObj:=wWobj;
    pTarget.trans := [7,29.0,0];
    MoveL pTarget,vSpeed,z0,tTool\WObj:=wWobj;
    pTarget.trans := [9,31.0,0];
    MoveL pTarget,vSpeed,z0,tTool\WObj:=wWobj;
    pTarget.trans := [12,32.0,0];
    MoveL pTarget,vSpeed,z0,tTool\WObj:=wWobj;
    pTarget.trans := [15,32.0,0];
    MoveL pTarget,vSpeed,z0,tTool\WObj:=wWobj;
    pTarget.trans := [17,31.0,0];
    MoveL pTarget,vSpeed,z0,tTool\WObj:=wWobj;
    pTarget.trans := [18,29.0,0];
    MoveL pTarget,vSpeed,z0,tTool\WObj:=wWobj;
    pTarget.trans := [18,25.0,0];
    MoveL pTarget,vSpeed,z0,tTool\WObj:=wWobj;
    pTarget.trans := [17,22.0,0];
    MoveL pTarget,vSpeed,z0,tTool\WObj:=wWobj;
    pTarget.trans := [15,19.0,0];
    MoveL pTarget,vSpeed,z0,tTool\WObj:=wWobj;
    pTarget.trans := [11,15.0,0];
    MoveL pTarget,vSpeed,z0,tTool\WObj:=wWobj;
    pTarget.trans := [8,13.0,0];
    MoveL pTarget,vSpeed,z0,tTool\WObj:=wWobj;
    pTarget.trans := [6,12.0,0];
    MoveL pTarget,vSpeed,z0,tTool\WObj:=wWobj;
    pTarget.trans := [3,11.0,0];
    MoveL pTarget,vSpeed,z0,tTool\WObj:=wWobj;
    pTarget.trans := [1,11.0,0];
    MoveL pTarget,vSpeed,z0,tTool\WObj:=wWobj;
    pTarget.trans := [0,12.0,0];
    MoveL pTarget,vSpeed,z0,tTool\WObj:=wWobj;
    pTarget.trans := [0,14.0,0];
    MoveL pTarget,vSpeed,z0,tTool\WObj:=wWobj;
    pTarget.trans := [1,15.0,0];
    MoveL pTarget,vSpeed,z0,tTool\WObj:=wWobj;
    pTarget.trans := [3,15.0,0];
    MoveL pTarget,vSpeed,z0,tTool\WObj:=wWobj;
    pTarget.trans := [5,14.0,0];
    MoveL pTarget,vSpeed,z0,tTool\WObj:=wWobj;
    pTarget.trans := [8,12.0,0];
    MoveL pTarget,vSpeed,z0,tTool\WObj:=wWobj;
    pTarget.trans := [11,11.0,0];
    MoveL pTarget,vSpeed,z0,tTool\WObj:=wWobj;
    pTarget.trans := [14,11.0,0];
    MoveL pTarget,vSpeed,z0,tTool\WObj:=wWobj;
    pTarget.trans := [17,12.0,0];
    MoveL pTarget,vSpeed,z0,tTool\WObj:=wWobj;
    pTarget.trans := [19,14.0,0];
    MoveL pTarget,vSpeed,fine,tTool\WObj:=wWobj;
    Reset do_pen;
    MoveL RelTool(pTarget,0,0,-2),vSpeed,z0,tTool\WObj:=wWobj;
    wWobj.oframe.trans.x := wWobj.oframe.trans.x + 19;
ENDPROC
  ! Character: R
  PROC char_upperR()
    VAR robtarget pTarget;
    pTarget := refTarget;
    pTarget.trans := [13,30.0,0];
    MoveL pTarget,vSpeed,fine,tTool\WObj:=wWobj;
    Set do_pen;
    pTarget.trans := [14,29.0,0];
    MoveL pTarget,vSpeed,z0,tTool\WObj:=wWobj;
    pTarget.trans := [14,26.0,0];
    MoveL pTarget,vSpeed,z0,tTool\WObj:=wWobj;
    pTarget.trans := [13,22.0,0];
    MoveL pTarget,vSpeed,z0,tTool\WObj:=wWobj;
    pTarget.trans := [12,19.0,0];
    MoveL pTarget,vSpeed,z0,tTool\WObj:=wWobj;
    pTarget.trans := [11,17.0,0];
    MoveL pTarget,vSpeed,z0,tTool\WObj:=wWobj;
    pTarget.trans := [9,14.0,0];
    MoveL pTarget,vSpeed,z0,tTool\WObj:=wWobj;
    pTarget.trans := [7,12.0,0];
    MoveL pTarget,vSpeed,z0,tTool\WObj:=wWobj;
    pTarget.trans := [5,11.0,0];
    MoveL pTarget,vSpeed,z0,tTool\WObj:=wWobj;
    pTarget.trans := [4,11.0,0];
    MoveL pTarget,vSpeed,z0,tTool\WObj:=wWobj;
    pTarget.trans := [3,12.0,0];
    MoveL pTarget,vSpeed,z0,tTool\WObj:=wWobj;
    pTarget.trans := [3,15.0,0];
    MoveL pTarget,vSpeed,z0,tTool\WObj:=wWobj;
    pTarget.trans := [4,20.0,0];
    MoveL pTarget,vSpeed,z0,tTool\WObj:=wWobj;
    pTarget.trans := [5,23.0,0];
    MoveL pTarget,vSpeed,z0,tTool\WObj:=wWobj;
    pTarget.trans := [6,25.0,0];
    MoveL pTarget,vSpeed,z0,tTool\WObj:=wWobj;
    pTarget.trans := [8,28.0,0];
    MoveL pTarget,vSpeed,z0,tTool\WObj:=wWobj;
    pTarget.trans := [10,30.0,0];
    MoveL pTarget,vSpeed,z0,tTool\WObj:=wWobj;
    pTarget.trans := [12,31.0,0];
    MoveL pTarget,vSpeed,z0,tTool\WObj:=wWobj;
    pTarget.trans := [15,32.0,0];
    MoveL pTarget,vSpeed,z0,tTool\WObj:=wWobj;
    pTarget.trans := [19,32.0,0];
    MoveL pTarget,vSpeed,z0,tTool\WObj:=wWobj;
    pTarget.trans := [21,31.0,0];
    MoveL pTarget,vSpeed,z0,tTool\WObj:=wWobj;
    pTarget.trans := [22,30.0,0];
    MoveL pTarget,vSpeed,z0,tTool\WObj:=wWobj;
    pTarget.trans := [23,28.0,0];
    MoveL pTarget,vSpeed,z0,tTool\WObj:=wWobj;
    pTarget.trans := [23,25.0,0];
    MoveL pTarget,vSpeed,z0,tTool\WObj:=wWobj;
    pTarget.trans := [22,23.0,0];
    MoveL pTarget,vSpeed,z0,tTool\WObj:=wWobj;
    pTarget.trans := [21,22.0,0];
    MoveL pTarget,vSpeed,z0,tTool\WObj:=wWobj;
    pTarget.trans := [19,21.0,0];
    MoveL pTarget,vSpeed,z0,tTool\WObj:=wWobj;
    pTarget.trans := [16,21.0,0];
    MoveL pTarget,vSpeed,z0,tTool\WObj:=wWobj;
    pTarget.trans := [13,22.0,0];
    MoveL pTarget,vSpeed,z0,tTool\WObj:=wWobj;
    pTarget.trans := [14,21.0,0];
    MoveL pTarget,vSpeed,z0,tTool\WObj:=wWobj;
    pTarget.trans := [15,19.0,0];
    MoveL pTarget,vSpeed,z0,tTool\WObj:=wWobj;
    pTarget.trans := [15,14.0,0];
    MoveL pTarget,vSpeed,z0,tTool\WObj:=wWobj;
    pTarget.trans := [16,12.0,0];
    MoveL pTarget,vSpeed,z0,tTool\WObj:=wWobj;
    pTarget.trans := [18,11.0,0];
    MoveL pTarget,vSpeed,z0,tTool\WObj:=wWobj;
    pTarget.trans := [20,12.0,0];
    MoveL pTarget,vSpeed,z0,tTool\WObj:=wWobj;
    pTarget.trans := [21,13.0,0];
    MoveL pTarget,vSpeed,z0,tTool\WObj:=wWobj;
    pTarget.trans := [23,16.0,0];
    MoveL pTarget,vSpeed,fine,tTool\WObj:=wWobj;
    Reset do_pen;
    MoveL RelTool(pTarget,0,0,-2),vSpeed,z0,tTool\WObj:=wWobj;
    wWobj.oframe.trans.x := wWobj.oframe.trans.x + 20;
ENDPROC
  ! Character: S
  PROC char_upperS()
    VAR robtarget pTarget;
    pTarget := refTarget;
    pTarget.trans := [0,11.0,0];
